IF 	eState = 0 THEN // eDisabled := 0,	
	sStateDesc := 'Wyłączona';
ELSIF 	eState = 1 THEN // eAborted := 1,
	sStateDesc := 'Bezpieczne zatrzymanie';
ELSIF 	eState = 2 THEN // eAborting := 2,  
	sStateDesc := 'Bezpieczne zatrzymywanie';
ELSIF 	eState = 3 THEN // eError := 3,	
	sStateDesc := 'Błąd';
ELSIF 	eState = 4 THEN // eResetting := 4,	
	sStateDesc := 'Resetowanie';
ELSIF 	eState = 5 THEN // eManualMovement := 5, 
	sStateDesc := 'Tryb serwisowy';
ELSIF 	eState = 6 THEN // eHoming := 6,
	sStateDesc := 'Bazowanie';
ELSIF 	eState = 7 THEN // eHomingDone := 7,
	sStateDesc := 'Koniec bazowania';	
ELSIF 	eState = 8 THEN // ePreparingToReady := 8,	
	sStateDesc := 'Przygotowanie do gotowości';
ELSIF 	eState = 9 THEN // ePreparingToDisable := 9,
	sStateDesc := 'Przygotowanie do wyłączenia';	
ELSIF 	eState = 10 THEN // eReady	:= 10,
	sStateDesc := 'Gotowa';	
ELSIF 	eState = 11 THEN // eStopping := 11,
	sStateDesc := 'Zatrzymywanie';	
ELSIF 	eState = 12 THEN // eStarting := 12,
	sStateDesc := 'Uruchamianie';  
ELSIF 	eState = 13 THEN // eRunning := 13		
	sStateDesc := 'Praca';
END_IF

IF eState = 13 OR bRun THEN
	GripperScrewer();
	BottleSorter();
	RollerScrewer();	
	EntranceGates();
	CatchStation();
	MassHeating();
	Conveyor();
	CapFeeder();
	Checker();
	Dispencer();
	DispencerLifter();
	Robot();
	Weight();
	WeightLift();
	Drag();
	DragPneum();
	LidFeeder();
	LidSealing();
	WickFeeder();
END_IF

iState := eState;

ACTION BottleSorter:

IF eBottleSorterRunningState  = 1 THEN 
	sStateDesc := 'Błąd';	
ELSIF eBottleSorterRunningState  = 2 THEN 
	sStateDesc := 'Gotowa';	
ELSIF eBottleSorterRunningState  = 3 THEN 
	sStateDesc := 'Bazowanie';	
ELSIF eBottleSorterRunningState  = 4 THEN 
	sStateDesc := 'Koniec bazowania';	
ELSIF eBottleSorterRunningState  = 5 THEN 
	sStateDesc := 'Tryb ręczny';
ELSIF eBottleSorterRunningState  = 60 THEN 
	sStateDesc := 'Przygotowanie do ruchu';	
ELSIF eBottleSorterRunningState  = 70 THEN 
	sStateDesc := 'Zamknięcie bramki lewej';	
ELSIF eBottleSorterRunningState  = 80 THEN 
	sStateDesc := 'Przejazd do pobrania';	
ELSIF eBottleSorterRunningState  = 90 THEN 
	sStateDesc := 'Zamykanie chwytaka';	
ELSIF eBottleSorterRunningState  = 100 THEN 
	sStateDesc := 'Otwarcie bramki prawej';	
ELSIF eBottleSorterRunningState  = 110 THEN 
	sStateDesc := 'Przejazd nad formatke';	
ELSIF eBottleSorterRunningState  = 120 THEN 
	sStateDesc := 'Zamknięcie bramki lewej';	
ELSIF eBottleSorterRunningState  = 130 THEN 
	sStateDesc := 'Zamknięcie docisku';	
ELSIF eBottleSorterRunningState  = 140 THEN 
	sStateDesc := 'Wkładanie opakowania';	
ELSIF eBottleSorterRunningState  = 150 THEN 
	sStateDesc := 'Otwieranie chwytaka';
ELSIF eBottleSorterRunningState  = 160 THEN 
	sStateDesc := 'Powrót do pozycji gotowości';
ELSIF eBottleSorterRunningState  = 170 THEN 
	sStateDesc := 'Wypuszczanie formatki';
		
END_IF
END_ACTION

ACTION CapFeeder:
IF eCapFeederRunningState = 1 THEN
	sStateDesc := 'Gotowy';
ELSIF eCapFeederRunningState = 2 THEN
	sStateDesc := 'Niski poziom zamknięć';
ELSIF eCapFeederRunningState = 3 THEN
	sStateDesc := 'Praca';
ELSIF eCapFeederRunningState = 4 THEN
	sStateDesc := 'Zapełniony';
END_IF
END_ACTION

ACTION CapPushing:
IF eCapPushingRunningState = 1 THEN
	sStateDesc := 'Gotowy';
ELSIF eCapPushingRunningState = 2 THEN
	sStateDesc := 'Wbijanie';
ELSIF eCapPushingRunningState = 3 THEN
	sStateDesc := 'Przyciskanie';	
ELSIF eCapPushingRunningState = 4 THEN
	sStateDesc := 'Wbito';		
ELSIF eCapPushingRunningState = 5 THEN
	sStateDesc := 'Podnoszenie';									
END_IF
END_ACTION

ACTION CatchStation:
IF eCatchRunningState = 1 THEN
	sStateDesc := 'Błąd';
ELSIF eCatchRunningState = 2 THEN
	sStateDesc := 'Tryb serwisowy';
ELSIF eCatchRunningState = 4 THEN
	sStateDesc := 'Bazowanie';	
ELSIF eCatchRunningState = 5 THEN
	sStateDesc := 'Koniec bazownia';		
ELSIF eCatchRunningState = 6 THEN
	sStateDesc := 'Gotowość';			
ELSIF eCatchRunningState = 7 THEN
	sStateDesc := 'Chwytanie';				
ELSIF eCatchRunningState = 8 THEN
	sStateDesc := 'Chwycono';					
ELSIF eCatchRunningState = 9 THEN
	sStateDesc := 'Przygotowanie do wyłączenia';	
ELSIF eCatchRunningState = 10 THEN
	sStateDesc := 'Nie chwycono';					
END_IF
END_ACTION

ACTION Checker:
IF eCheckerRunningState = 1 THEN
	sStateDesc := 'Blad';
ELSIF eCheckerRunningState = 2 THEN
	sStateDesc := 'Tryb serwisowy';	
ELSIF eCheckerRunningState = 3 THEN
	sStateDesc := 'Bazowanie';		
ELSIF eCheckerRunningState = 4 THEN
	sStateDesc := 'Koniec bazowania';			
ELSIF eCheckerRunningState = 5 THEN
	sStateDesc := 'Gotowa';				
ELSIF eCheckerRunningState = 6 THEN
	sStateDesc := 'Formatka';		
ELSIF eCheckerRunningState = 7 THEN
	sStateDesc := 'Butelka';	
ELSIF eCheckerRunningState = 8 THEN
	sStateDesc := 'Platynka OK';	
ELSIF eCheckerRunningState = 9 THEN
	sStateDesc := 'Nasadka OK';	
ELSIF eCheckerRunningState = 10 THEN
	sStateDesc := 'Nasadka NOK.';		
ELSIF eCheckerRunningState = 11 THEN
	sStateDesc := 'Przyg. do wył.';		
					
END_IF
END_ACTION

ACTION Conveyor:
(*IF eConveyorRunningState = 0 THEN //Wyłączona
	sStateDesc := 'Wyłączona';
ELSIF eConveyorRunningState = 1 THEN //Błąd
	sStateDesc := 'Bład';
ELSIF eConveyorRunningState = 2 THEN //Tryb serwisowy
	sStateDesc := 'Tryb serwisowy';	
ELSIF eConveyorRunningState = 3 THEN //Bazowanie
	sStateDesc := 'Bazowanie';		
ELSIF eConveyorRunningState = 4 THEN //Koniec bazowania
	sStateDesc := 'Koniec bazowanie';	
ELSIF eConveyorRunningState = 5 THEN //gotowość
	sStateDesc := 'Gotowa';	
ELSIF eConveyorRunningState = 6 THEN //Zatrzymywanie
	sStateDesc := 'Zatrzymywanie';	
ELSIF eConveyorRunningState = 7 THEN //Startowanie
	sStateDesc := 'Startowanie';	
ELSIF eConveyorRunningState = 8 THEN //Praca
	sStateDesc := 'Praca';				
END_IF


*)
(*
IF eConveyorRunningState = 0 THEN //Wyłączona
	sStateDesc := 'Wyłączona 123';
ELSIF eConveyorRunningState = 1 THEN //Błąd
	sStateDesc := 'Bezp. zatrzymana';
ELSIF eConveyorRunningState = 2 THEN //Tryb serwisowy
	sStateDesc := 'Bezp. zatrzymywanie';	
ELSIF eConveyorRunningState = 3 THEN //Bazowanie
	sStateDesc := 'Błąd';		
ELSIF eConveyorRunningState = 4 THEN //Koniec bazowania
	sStateDesc := 'Resetowanie błędów';	
ELSIF eConveyorRunningState = 5 THEN //gotowość
	sStateDesc := 'Tryb ręczny';	
ELSIF eConveyorRunningState = 6 THEN //Zatrzymywanie
	sStateDesc := 'Bazowanie';	
ELSIF eConveyorRunningState = 7 THEN //Startowanie
	sStateDesc := 'Koniec bazowania';	
ELSIF eConveyorRunningState = 8 THEN //Praca
	sStateDesc := 'Przyg. do wył.';	
	*)
IF eConveyorRunningState = 10 THEN //Startowanie
	sStateDesc := 'Gotowośc';	
ELSIF eConveyorRunningState = 11 THEN //Praca
	sStateDesc := 'Zatrzymywanie';	
ELSIF eConveyorRunningState = 12 THEN //Praca
	sStateDesc := 'Uruchamianie';	
ELSIF eConveyorRunningState = 13 THEN //Praca
	sStateDesc := 'Praca';

	
END_IF
END_ACTION

ACTION Dispencer:
IF eDispencerRunningState = 5 THEN
	sStateDesc := 'Gotowa';	
		ic3		:= ic3+1;		
ELSIF eDispencerRunningState = 6 THEN
	sStateDesc := 'Przyg. dozy';		
ELSIF eDispencerRunningState = 7 THEN
	sStateDesc := '1 faza';	
ELSIF eDispencerRunningState = 8 THEN
	sStateDesc := '2 faza';	
ELSIF eDispencerRunningState = 9 THEN
	sStateDesc := '3 faza';	
ELSIF eDispencerRunningState = 10 THEN
	sStateDesc := 'Koniec dozy';	
ELSIF eDispencerRunningState = 11 THEN
	sStateDesc := 'Podsys';	
ELSIF eDispencerRunningState = 12 THEN
	sStateDesc := 'Koniec pods.';	
ELSIF eDispencerRunningState = 13 THEN
	sStateDesc := 'Zasysanie';				
ELSIF eDispencerRunningState = 14 THEN
	sStateDesc := 'Podnoszenie';	
ELSIF eDispencerRunningState = 15 THEN
	sStateDesc := 'Przerywanie';			
ELSIF eDispencerRunningState = 16 THEN
	sStateDesc := 'Przyg. do wył.';	
ELSIF eDispencerRunningState = 17 THEN
	sStateDesc := 'Przeciąganie';
ELSIF eDispencerRunningState = 18 THEN
	sStateDesc := 'Przyg. do mycia';
ELSIF eDispencerRunningState = 19 THEN
	sStateDesc := 'Gotowy do mycia';
ELSIF eDispencerRunningState = 20 THEN
	sStateDesc := 'Mycie';
ELSIF eDispencerRunningState = 21 THEN
	sStateDesc := 'Koniec mycia';		
END_IF

i   := eDispencerRunningState;
END_ACTION

ACTION DispencerLifter:
IF eDispencerLifterRunningState = 1 THEN
	sStateDesc := 'Blad';
ELSIF eDispencerLifterRunningState = 2 THEN
	sStateDesc := 'Tryb serwisowy';	
ELSIF eDispencerLifterRunningState = 3 THEN
	sStateDesc := 'Bazowanie';		
ELSIF eDispencerLifterRunningState = 4 THEN
	sStateDesc := 'Koniec bazowania';			
ELSIF eDispencerLifterRunningState = 5 THEN
	sStateDesc := 'Gotowa';				
ELSIF eDispencerLifterRunningState = 6 THEN
	sStateDesc := 'Przyg. dozy';		
ELSIF eDispencerLifterRunningState = 7 THEN
	sStateDesc := '1 faza';	
ELSIF eDispencerLifterRunningState = 8 THEN
	sStateDesc := '2 faza';	
ELSIF eDispencerLifterRunningState = 9 THEN
	sStateDesc := '3 faza';	
ELSIF eDispencerLifterRunningState = 10 THEN
	sStateDesc := 'Koniec dozy';	
ELSIF eDispencerLifterRunningState = 11 THEN
	sStateDesc := 'Zasysanie';	
ELSIF eDispencerLifterRunningState = 12 THEN
	sStateDesc := 'Podnoszenie';	
ELSIF eDispencerLifterRunningState = 13 THEN
	sStateDesc := 'Wylaczanie';				
ELSIF eDispencerLifterRunningState = 14 THEN
	sStateDesc := 'Przyg. do wył.';	
ELSIF eDispencerLifterRunningState = 15 THEN
	sStateDesc := 'Przeciąganie';			
ELSIF eDispencerLifterRunningState = 16 THEN
	sStateDesc := 'Podsysanie';	
ELSIF eDispencerLifterRunningState = 17 THEN
	sStateDesc := 'Koniec podsysania';		
END_IF
END_ACTION

ACTION Drag:
IF eFormsDragingRunningState = 1 THEN 
	sStateDesc := 'Bład';
ELSIF eFormsDragingRunningState  = 2 THEN 
	sStateDesc := 'Gotowość';	
ELSIF eFormsDragingRunningState  = 3 THEN 
	sStateDesc := 'Tryb serwisowy';	
ELSIF eFormsDragingRunningState  = 4 THEN 
	sStateDesc := 'Przygotowanie do ruchu';	
ELSIF eFormsDragingRunningState  = 5 THEN 
	sStateDesc := 'Bazowanie';	
ELSIF eFormsDragingRunningState  = 6 THEN 
	sStateDesc := 'Koniec bazowania';	
ELSIF eFormsDragingRunningState  = 7 THEN 
	sStateDesc := 'Podnoszenie';	
ELSIF eFormsDragingRunningState  = 8 THEN 
	sStateDesc := 'Przyg. do przec.';	
ELSIF eFormsDragingRunningState  = 9 THEN 
	sStateDesc := 'Przeciąganie';	
ELSIF eFormsDragingRunningState  = 10 THEN 
	sStateDesc := 'Koniec Przec.';	
ELSIF eFormsDragingRunningState  = 11 THEN 
	sStateDesc := 'Zakańczanie przec.';	
ELSIF eFormsDragingRunningState  = 12 THEN 
	sStateDesc := 'Koniec zakań. przec.';	
ELSIF eFormsDragingRunningState  = 13 THEN 
	sStateDesc := 'Opuszczanie';	
ELSIF eFormsDragingRunningState  = 14 THEN 
	sStateDesc := 'Przeciągniete';	
ELSIF eFormsDragingRunningState  = 15 THEN 
	sStateDesc := 'Koniec cyklu';	
			
END_IF
END_ACTION

ACTION DragPneum:
IF eFormsDragingPneumRunningState= 1 THEN 
	sStateDesc := 'Bład';
ELSIF eFormsDragingPneumRunningState  = 2 THEN 
	sStateDesc := 'Gotowość';	
ELSIF eFormsDragingPneumRunningState  = 3 THEN 
	sStateDesc := 'Tryb serwisowy';	
ELSIF eFormsDragingPneumRunningState  = 4 THEN 
	sStateDesc := 'Przygotowanie do ruchu';	
ELSIF eFormsDragingPneumRunningState  = 5 THEN 
	sStateDesc := 'Bazowanie';	
ELSIF eFormsDragingPneumRunningState  = 6 THEN 
	sStateDesc := 'Koniec bazowania';	
ELSIF eFormsDragingPneumRunningState  = 7 THEN 
	sStateDesc := 'Podnoszenie';	
ELSIF eFormsDragingPneumRunningState  = 8 THEN 
	sStateDesc := 'Przyg. do przec.';	
ELSIF eFormsDragingPneumRunningState  = 9 THEN 
	sStateDesc := 'Przeciąganie';	
ELSIF eFormsDragingPneumRunningState  = 10 THEN 
	sStateDesc := 'Koniec Przec.';	
ELSIF eFormsDragingPneumRunningState  = 11 THEN 
	sStateDesc := 'Korekta pozycji';	
ELSIF eFormsDragingPneumRunningState  = 12 THEN 
	sStateDesc := 'Koniec korekty';	
ELSIF eFormsDragingPneumRunningState  = 13 THEN 
	sStateDesc := 'Opuszczanie';	
ELSIF eFormsDragingPneumRunningState  = 14 THEN 
	sStateDesc := 'Przeciągniete';	
ELSIF eFormsDragingPneumRunningState  = 15 THEN 
	sStateDesc := 'Koniec cyklu';					
END_IF
END_ACTION

ACTION EntranceGates:
IF eEntranceGatesRunningState = 1 THEN
	sStateDesc := 'Błąd';
ELSIF eEntranceGatesRunningState = 2 THEN
	sStateDesc := 'Tryb serwisowy';
ELSIF eEntranceGatesRunningState = 4 THEN
	sStateDesc := 'Bazowanie';	
ELSIF eEntranceGatesRunningState = 5 THEN
	sStateDesc := 'Koniec bazownia';		
ELSIF eEntranceGatesRunningState = 6 THEN
	sStateDesc := 'Gotowość';			
ELSIF eEntranceGatesRunningState = 8 THEN
	sStateDesc := 'Wjazd 2 ';				
ELSIF eEntranceGatesRunningState = 9 THEN
	sStateDesc := 'Wjazd 1';					
ELSIF eEntranceGatesRunningState = 11 THEN
	sStateDesc := 'Czekanie';						
ELSIF eEntranceGatesRunningState = 12 THEN
	sStateDesc := 'Wyjazd 2';							
ELSIF eEntranceGatesRunningState = 13 THEN
	sStateDesc := 'Wyjazd 1';	
ELSIF eEntranceGatesRunningState = 14 THEN
	sStateDesc := 'Blokowanie';	
ELSIF eEntranceGatesRunningState = 15 THEN
	sStateDesc := 'Otwieranie';	
ELSIF eEntranceGatesRunningState = 16 THEN
	sStateDesc := 'Otwarty';	
ELSIF eEntranceGatesRunningState = 17 THEN
	sStateDesc := 'Przygotowanie do gotowości';	
ELSIF eEntranceGatesRunningState = 18 THEN
	sStateDesc := 'Przygotowanie do wyłączenia';	
ELSIF eEntranceGatesRunningState = 19 THEN
	sStateDesc := 'Przeciąganie do środka';	
ELSIF eEntranceGatesRunningState = 20 THEN
	sStateDesc := 'Przeciągnięto do środka';			
END_IF
END_ACTION

ACTION GripperScrewer:
IF eGripperScrewerRunningState = 1 THEN
	sStateDesc := 'Gotowa';
ELSIF eGripperScrewerRunningState = 2 THEN
	sStateDesc := 'Przejazd do wbijania';
ELSIF eGripperScrewerRunningState = 3 THEN
	sStateDesc := 'Przejazd do zakrecania';	
ELSIF eGripperScrewerRunningState = 4 THEN
	sStateDesc := 'Wcisnieto';		
ELSIF eGripperScrewerRunningState = 5 THEN
	sStateDesc := 'Szukanie gwintu';			
ELSIF eGripperScrewerRunningState = 6 THEN
	sStateDesc := 'Zakrecanie';				
ELSIF eGripperScrewerRunningState = 7 THEN
	sStateDesc := 'Podnoszenie';					
ELSIF eGripperScrewerRunningState = 8 THEN
	sStateDesc := 'Zakrecono';						
ELSIF eGripperScrewerRunningState = 9 THEN
	sStateDesc := 'Niezakręcono';							
ELSIF eGripperScrewerRunningState = 10 THEN
	sStateDesc := 'Przytrzymywanie';			
END_IF
END_ACTION

ACTION LidFeeder:
IF eLidFeederRunningState = 1 THEN
	sStateDesc := 'Blad';
ELSIF eLidFeederRunningState = 2 THEN
	sStateDesc := 'Tryb serwisowy';	
ELSIF eLidFeederRunningState = 3 THEN
	sStateDesc := 'Bazowanie';		
ELSIF eLidFeederRunningState = 4 THEN
	sStateDesc := 'Koniec bazowania';			
ELSIF eLidFeederRunningState = 5 THEN
	sStateDesc := 'Nagrzewanie';				
ELSIF eLidFeederRunningState = 6 THEN
	sStateDesc := 'Gotowa';		
ELSIF eLidFeederRunningState = 7 THEN
	sStateDesc := 'Zasysanie';	
ELSIF eLidFeederRunningState = 8 THEN
	sStateDesc := 'Nakładanie';	
ELSIF eLidFeederRunningState = 9 THEN
	sStateDesc := 'Nakładanie 2';	
ELSIF eLidFeederRunningState = 10 THEN
	sStateDesc := 'Zgrzewanie';	
ELSIF eLidFeederRunningState = 11 THEN
	sStateDesc := 'Odlożona';	
ELSIF eLidFeederRunningState = 12 THEN
	sStateDesc := 'Podnoszenie';	
ELSIF eLidFeederRunningState = 13 THEN
	sStateDesc := 'Przyg.do wyłączenia';						
END_IF
END_ACTION

ACTION LidSealing:

IF eLidSealingRunningState = 1 THEN
	sStateDesc := 'Nagrzewanie';
ELSIF eLidSealingRunningState = 2 THEN
	sStateDesc := 'Gotowa';	
ELSIF eLidSealingRunningState = 3 THEN
	sStateDesc := 'Zgrzewanie';		
ELSIF eLidSealingRunningState = 4 THEN
	sStateDesc := 'Grzanie';			
ELSIF eLidSealingRunningState = 5 THEN
	sStateDesc := 'Zgrzano';				
ELSIF eLidSealingRunningState = 6 THEN
	sStateDesc := 'Podnoszenie';							
END_IF
END_ACTION

ACTION MassHeating:
IF eMassHeatingRunningState = 1 THEN //Grzanie
	sStateDesc := 'Grzanie';
ELSIF eMassHeatingRunningState = 2 THEN //Gotowość
	sStateDesc := 'Utrzymywanie temp.';	
ELSIF eMassHeatingRunningState = 3 THEN //Chłodzenie
	sStateDesc := 'Chłodzenie';					
END_IF
END_ACTION

ACTION Robot:
IF eCapFeederRobotRunningState = 1 THEN
	sStateDesc := 'Pobieranie';
ELSIF eCapFeederRobotRunningState = 2 THEN
	sStateDesc := 'Pobrano';
ELSIF eCapFeederRobotRunningState = 3 THEN
	sStateDesc := 'Odkładanie';	
ELSIF eCapFeederRobotRunningState = 4 THEN
	sStateDesc := 'Pobrano';		
ELSIF eCapFeederRobotRunningState = 5 THEN
	sStateDesc := 'Odrzucanie';			
ELSIF eCapFeederRobotRunningState = 6 THEN
	sStateDesc := 'Odrzucono';				
ELSIF eCapFeederRobotRunningState = 7 THEN
	sStateDesc := 'Do start Inkjet';	
ELSIF eCapFeederRobotRunningState = 8 THEN
	sStateDesc := 'Start Inkjet';		
ELSIF eCapFeederRobotRunningState = 9 THEN
	sStateDesc := 'Do stop Inkjet';		
ELSIF eCapFeederRobotRunningState = 10 THEN
	sStateDesc := 'Stop Inkjet';		
ELSIF eCapFeederRobotRunningState = 11 THEN
	sStateDesc := 'Przerywanie';		
ELSIF eCapFeederRobotRunningState = 12 THEN
	sStateDesc := 'Powrót do gotowości';		
ELSIF eCapFeederRobotRunningState = 13 THEN
	sStateDesc := 'Pobieranie po Estopie';						
END_IF
END_ACTION

ACTION RollerScrewer:
(*IF eRollerScrewerRunningState = 1 THEN
	sStateDesc := 'Gotowa';
ELSIF eRollerScrewerRunningState = 2 THEN
	sStateDesc := 'Wciskanie';
ELSIF eRollerScrewerRunningState = 3 THEN
	sStateDesc := '';	
ELSIF eRollerScrewerRunningState = 4 THEN
	sStateDesc := 'Wcisnieto';		
ELSIF eRollerScrewerRunningState = 5 THEN
	sStateDesc := 'Szukanie gwintu';			
ELSIF eRollerScrewerRunningState = 6 THEN
	sStateDesc := 'Zakrecanie';				
ELSIF eRollerScrewerRunningState = 7 THEN
	sStateDesc := 'Podnoszenie';					
ELSIF eRollerScrewerRunningState = 8 THEN
	sStateDesc := 'Zakrecono';						
ELSIF eRollerScrewerRunningState = 9 THEN
	sStateDesc := 'Niezakręcono';							
ELSIF eRollerScrewerRunningState = 10 THEN
	sStateDesc := 'Przytrzymywanie';			
END_IF

*)
END_ACTION

ACTION Weight:
IF  eWeightRunningState = 1 THEN
	sStateDesc := 'Gotowa';	
ELSIF eWeightRunningState = 2 THEN
	sStateDesc := 'Ważenie';		
ELSIF eWeightRunningState = 3 THEN
	sStateDesc := 'Koniec ważenia';					
END_IF
END_ACTION

ACTION WeightLift:
IF  eWeightLiftRunningState	 = 10 THEN
	sStateDesc := 'Gotowa';	
ELSIF eWeightLiftRunningState	= 20 THEN
	sStateDesc := 'Przyg do magazynowania formatek';		
ELSIF eWeightLiftRunningState	 = 30 THEN
	sStateDesc := 'Czekanie na formatki';		
ELSIF eWeightLiftRunningState	 = 40 THEN
	sStateDesc := 'Rozpoczęcie ważenia';		
ELSIF eWeightLiftRunningState	 = 50 THEN
	sStateDesc := 'Ważenie';		
ELSIF eWeightLiftRunningState	 = 60 THEN
	sStateDesc := 'Opuszczanie wideł';		
ELSIF eWeightLiftRunningState	 = 70 THEN
	sStateDesc := 'Wypuszczanie formatek';		
ELSIF eWeightLiftRunningState	 = 80 THEN
	sStateDesc := 'Cykl skończony';			
END_IF
END_ACTION

ACTION Wheel:
(*IF eWheelRunningState = 1 THEN
	sStateDesc := 'Blad';
ELSIF eWheelRunningState = 2 THEN
	sStateDesc := 'Tryb serwisowy';	
ELSIF eWheelRunningState = 3 THEN
	sStateDesc := 'Bazowanie';		
ELSIF eWheelRunningState = 4 THEN
	sStateDesc := 'Koniec bazowania';			
ELSIF eWheelRunningState = 5 THEN
	sStateDesc := 'Gotowa';				
ELSIF eWheelRunningState = 6 THEN
	sStateDesc := 'Obracanie';		
ELSIF eWheelRunningState = 7 THEN
	sStateDesc := 'Koniec obracania';	
ELSIF eWheelRunningState = 8 THEN
	sStateDesc := 'Przerywanie';	
ELSIF eWheelRunningState = 9 THEN
	sStateDesc := 'Obracanie 2';	
ELSIF eWheelRunningState = 10 THEN
	sStateDesc := 'Przygtowanie go obr.';						
END_IF
*)
END_ACTION

ACTION WickFeeder:
IF eWickFeederRunningState = 1 THEN
	sStateDesc := 'Blad';
ELSIF eWickFeederRunningState = 2 THEN
	sStateDesc := 'Tryb serwisowy';	
ELSIF eWickFeederRunningState = 3 THEN
	sStateDesc := 'Bazowanie';		
ELSIF eWickFeederRunningState = 4 THEN
	sStateDesc := 'Koniec bazowania';			
ELSIF eWickFeederRunningState = 5 THEN
	sStateDesc := 'Nagrzewanie';				
ELSIF eWickFeederRunningState = 6 THEN
	sStateDesc := 'Gotowa';		
ELSIF eWickFeederRunningState = 7 THEN
	sStateDesc := 'Zasysanie';	
ELSIF eWickFeederRunningState = 8 THEN
	sStateDesc := 'Nakładanie';	
ELSIF eWickFeederRunningState = 9 THEN
	sStateDesc := 'Nakładanie 2';	
ELSIF eWickFeederRunningState = 10 THEN
	sStateDesc := 'Zgrzewanie';	
ELSIF eWickFeederRunningState = 11 THEN
	sStateDesc := 'Odlożona';	
ELSIF eWickFeederRunningState = 12 THEN
	sStateDesc := 'Podnoszenie';	
ELSIF eWickFeederRunningState = 13 THEN
	sStateDesc := 'Przyg.do wyłączenia';						
END_IF
END_ACTION

END_FUNCTION_BLOCK

// ---- POUs/FB/FB_ROPPFeeder.TcPOU
(*
Nazwa:			FB_ROPPFeeder
Opis:			Sorter nasadek i podajnik nasadek z podnośnikiem JIESANG
Wersja:			v0.1
Data:			2022-07-07
Autor:			DJA
Urzadzenia:		Silnik sortera, podnośnik JIESANG, Wydmuch, czujniki zapełnienia rękawa
Konfiguracja:	
Info:
-poprawiona wersja sortera względem poprzedniej, przerobione na aktualny standard State i RunningState
*)


FUNCTION_BLOCK FB_ROPPFeeder
VAR_INPUT
	
	bEnable						: BOOL;					//Zezowlenie na pracę stacji sprawdzania
	bEStop						: BOOL;					//Stop Awaryjny nieaktywny
	bRun						: BOOL;					//
	bHoming						: BOOL;					//Zezwolenie na wykonanie bazowania i pozycjonowania stacji sprawdzania
	bHeightSet					: BOOL;					//Bit do bazowania stacji na ustaloną wysokość 
	bIgnoreError				: BOOL;					//Ignorowania błędów cyklu pracy
	bReset						: BOOL;					//Reset błędu, jeśli w stanie "eError"

	bConveyorOKSensor			: BOOL;					
	bConveyorNOKSensor			: BOOL;				
	bAirOKSensor				: BOOL;					// 
	bCapsWheelLevelSensor		: BOOL;					// Czujnik poziomu
	bCapsLevelSensor			: BOOL;					// Czujnik poziomu
	bCapsSleeveSensor			: BOOL;					// 

	iTimeDelayOn				: INT; 					//Czas na właczenie silnika sortera po zaniku sygnału przepełnienia z rękawa
	iTimeDelayOff				: INT; 					// Czas na wylączenie silnika sortera po wykryciu sygnału przepełnienia z rękawa sortera
	iTimeToEmptySleeveError		: INT;					// Czas do włączenia alrmu pustego rękawa
	InEngineVelocityCV 			: UDINT;		
	InEngineSTW 				: UINT; 				// Statusword transportera wejściowo wyjściowego
	IbEngineWcState				: BOOL; 				// Statusword transportera wejściowo wyjściowego

	_HEIGHTMOTOR_ 				: BOOL;
	lrHeightMotorSV				: LREAL;				// Zadana wysokość
	udiHeightMotorEncoderCV		: UDINT;				// Ilość impulsów z modułu enkoderowego
	bHeightEncoderSetCDone		: BOOL;					// Zerowanie enkodera wykonane
	rHeightMotorPositionOffset 	: REAL;					// Wysokość bazowani podnośnika
	lrMaxHeight					: LREAL;				// Maksymalna wysokość podnośnika chwytaka
	lrMinHeight					: LREAL;				// Minimalna wysokość podnośnika chwytaka

	bManualMovement				: BOOL; 				//Uruchomienie trybu ruchów ręcznych
	udiStationIndex				: UDINT;				// Indywidualny numer stacji
	sStationName				: STRING;				// Nazwa stacji	
END_VAR

VAR_OUTPUT
	eState						: E_Station;			// Aktualny stan stacju
	eRunningState				: E_CapFeederState;		// Stan pracy stacji
	eRunningStateBeforeEstop	: E_CapFeederState;  	// Stan przed Estope
	bError						: BOOL;					// Błąd stacji
	udiErrorID					: UDINT;				// Nr blędu przeciągania formatek
	sErrorDescription			: STRING(200);			// Opis błędu
	sErrorDescription2			: STRING(200);			// Opis błędu
	sErrorStationName			: STRING;				// Nazwa stacj
	udiStationID				: UDINT;				// Nr stacji

	bHeightMotorUp				: BOOL;					//Sterowanie silnikiem podnośnika  - RUCH W GÓRĘ
	bHeightMotorDown			: BOOL;					//Sterowanie silnikiem podnośnika  - RUCH W DÓŁ
	udiHeightMotorEncoderSetCV	: UDINT;		
	bHeightEncoderSetC			: BOOL;					// Zerowanie enkodera
	lrHeightMotorCV				: LREAL;				// Aktualna pozycja podnośnika

	QnEngineVelocitySV 			: UDINT; 				// Nastawa prędkości
	QnEngineCTW 				: UINT;  				// Controlword transportera we/wy	
	bSorterVibrator				: BOOL; 	
	bSorterAir 					: BOOL; 				
	bSorterAir2					: BOOL; 				
	bConveyorStart				: BOOL; 				
	bConveyorStop				: BOOL; 	
	
	bHomingNeeded				: BOOL;					// Wymagane ponowne bazowanie (blad podczas bazowania lub stop awaryjny)
	bHomingDone					: BOOL;					// Stacja zbazowana 
	bCycleDone					: BOOL;					// Sygnał o zakończeniu cyklu
	bCycleNotDone				: BOOL;					// Sygnał o niezakończonym cyklu
	tCycleTime					: TIME;	 				// Czas cyklu 
	sWarningDescription			: STRING;
	bWarning1					: BOOL;
	udiWarningID				: UDINT;
	
END_VAR

VAR_IN_OUT
	bManualHeightMotorUp		: BOOL;					//Ruch ręczny podnośnika stacji w górę
	bManualHeightMotorDown		: BOOL;					//Ruch ręczny podnośnika stacji w dół
	bManualSorterEngine			: BOOL;					//
	bManualSorterVibrator		: BOOL;					//
	bManualSorterAir 			: BOOL;					//
	bManualSorterAir2			: BOOL;					//
	bManualConveyorStart		: BOOL;					//
	bManualConveyorStop			: BOOL;					//
END_VAR

VAR
	i							:	INT;
	aBufferedSensorValue		:	ARRAY[0..50] OF BOOL;	
	rtOutSensor					:	R_TRIG;

	// State
	eLastState					: E_Station;			//Stan ogólny bloku
	eLastStateTemp				: E_Station;			//Stan ogólny bloku
	eLastRunningState			: E_CapFeederState;		//Stan podbloku
	eLastRunningStateTemp		: E_CapFeederState;		//Stan podbloku

	fbHeightMotorEncoder		: FB_JiesangActuatorEncoderModul;				// Blok enkodera podnośnika chwytaka stabilizującego pod zakręcarką	
	bHeightMotorEncoderCounterReset						:BOOL; 				// Sygnał resetu enkodera
	lrLastHeightMotorPositionCV		: LREAL;				// Pozycja podnośnika w poprzednim cyklu programu
	bHeightMotorEncoderHomed	: BOOL;					// Informacja od enkodera że jest zbazowany		
	bStateError					: BOOL;
	
	tofHeightMotorDown			: TOF;					// Opóźnienie ruchu w dół, żeby nie przeciązać rozruchem układu
	rtEncoderHomed				: R_TRIG;				// Bit zakończenia enkodera
		
	tonHeightNoChange			: TON; 					// Timer wykrycia braku ruchu siłownika zmiany wysokości stacji
	tonHeightNoChangeTime		: TON; 					// Timer wykrycia braku ruchu siłownika zmiany wysokości stacji
	
	tonLimitPosMinReachedDelay	: TON;					// Timer osoiągniecia minimalnej wyskości 
	tonLimitPosMaxReachedDelay	: TON;					// Timer osiągnięcia maksymalnej wyskości
	tonSortingEngineOn			: TON;					// Opóźnienie po załączeniu napędu
	tonSortingEngineOff			: TON;					// Opóźnienie wyłączenia napędu
	tonSleeveFullEngineOn		: TON;					// Czas załączenia napędu po wykrciu braku nasadek
	tonEngineBlocked			: TON;					// Zablokowany silnik	
	rtCapSorterSensor			: R_TRIG;				// Triger
	tonTryUnblockWheel			: TON;					// Czas ruchu falownika w drugą stronę
	tofCapFeederSorterCapSensor	: TOF;					// Opóźnienie sygnału z czujnika obecności nasadki ultradzwiek
	tonCapFeederSorterCapSensor	: TON;					// Opóźnienie sygnału z czujnika obecności nasadki ultradźwięk
	tonAirBeforeStart			: TON;					// Czasówka opóźeniani przedmuchu
	tonAirBeforeStart2			: TON;					// Czasówka opóźeniani przedmuchu
	tonAirAfterStop				: TON;					// Czasówka przedmuchu po zatrzymaniu
	tonStoppingTime				: TON;					// Czasówka zbyt długiego zatrzymawania

	
	tonErrorHeightChange		: TON; 					// Timer błędu zacięcia się podnośnika
	tonEmptySleeveError			: TON;					// Timer pustego rękawa
	tonMaxHeightError			: TON;					// Timer ustawienia zbyt dużej wysokości stacji
	tonMinHeightError			: TON;					// Timer ustawienia zbyt małej wysokości stacji
	tonCycleTimer				: TON;					// Czasówka cyklu
	rtrigCycleTimerRead			: R_TRIG;				// Trigger do statystyk cyklu 
	
	tonSorterEngineError: TON;

	TimerOn: TON;
	TimerOff: TON;
	bImpOn: BOOL;
	rtCapFeederSorterCapSensor: R_TRIG;
	bBlowDelay: BOOL;
	tonbBlowDelay: TON;
	
	fbInverter: FB_MitsubishiInverter;
	
	tonInverterError: TON;
	(*Ostrzeżenia*)
	fbbLevelSensor:	FB_InputFilter;
	(*Inne*)	
	fbbCapsWheelLevelSensor 		:	FB_InputFilter_v2;
	fbbCapsLevelSensor				:	FB_InputFilter_v2;


	tonGates1	:	TON;	//Czasówka dla szlabanów w rękawe
	tonGates2	:	TON;	//Czasówka dla szlabanów w rękawe
	tonGates3	:	TON;	//Czasówka dla szlabanów w rękawe
	tonGates4	:	TON;	//Czasówka dla szlabanów w rękawe

		
	bGates	    :	BOOL;	//Controla szłabanow w rękawe  
	bTryUnblockWheel : BOOL;
	iTryUnblockWheel : INT;
END_VAR

//Wywołanie bloczków od stacji. Ważna jest ich kolejność!!!
ACT_Limits();
ACT_HeightMotor();
ACT_ErrorHandling();

ACT_Signals();
ACT_Control();
ACT_Inverter();
ACT_Statistic();
ACT_Status();
ACT_Warnings();
aStationID();	

lrLastHeightMotorPositionCV:=lrHeightMotorCV;

ACTION ACT_Control:
	(*****Wyłączenie enable*****)
	IF NOT bEnable THEN
		IF eState <> E_Station.eDisabled AND eState <> E_Station.ePreparingToDisable THEN
				eState 				:= E_Station.ePreparingToDisable; 
		END_IF	
	END_IF

	(*****Estop*****)
	IF NOT bEstop  THEN	
		IF eState <> E_Station.eAborted AND eState <> E_Station.eAborting AND eState <> E_Station.eDisabled THEN
				eState 				:= E_Station.eAborting; 
		END_IF
	END_IF


	CASE eState OF
//--------------------------------------------------------------------------------
// Stan maszyny po wyłączeniu i przygotowanie do uruchomienia
	E_Station.eDisabled: 					// Stan nieaktywnosci (Stacja wyłączona) 
	
		IF bEnable THEN
			eState 				:= E_Station.ePreparingToReady; 
		END_IF 
		
//--------------------------------------------------------------------------------
// Stan maszyny po zatrzymaniu awaryjnym   
	E_Station.eAborted: 					// Stan bezpiecznego zatrzymania (po Abortingu) 

		IF bEStop THEN
			eState 				:= E_Station.ePreparingToReady;
		END_IF
		
//--------------------------------------------------------------------------------
// Stan maszyny naciśnieciu estopa 	
	E_Station.eAborting:                 	// Stan bezpiecznego zatrzymywania (po EStopie)

		ACT_ResetCommands();

		eState 						:=  E_Station.eAborted;  
		eRunningState				:=	E_CapFeederState.eReady;
		
//--------------------------------------------------------------------------------
// Stan masyzny po wykryciu błędu			
	E_Station.eError:                 	 	// Stan błędu 	
		
		ACT_ResetCommands();
		
		IF bReset THEN
			eState 				:= E_Station.eResetting;
			bError				:= FALSE;
		END_IF
		
//--------------------------------------------------------------------------------
// Stan masyzny po wykryciu błędu
	E_Station.eResetting:					// Stan resetowania bledu (po Errorze)
			CASE udiErrorID(*-udiStationIndex*) OF
		
				//Error 8 - Błąd falownika
				344:
					fbInverter.bReset	:= TRUE;
					bError 				:= FALSE;
				ELSE
					bError := FALSE;	
			END_CASE		
		
		IF NOT bError AND fbInverter.eState = E_Station.eReady THEN
			fbInverter.bReset	:= FALSE;	
			//{warning 'Sprawdzić błąd falownika CapFeeder'}
			udiErrorID 			:=	0;
			sErrorDescription 	:=	'';
			eState 				:=	E_Station.ePreparingToReady;
			eRunningState		:=	E_CapFeederState.eReady;
		ELSE
			eState 				:=	E_Station.eError;
		END_IF
    
//--------------------------------------------------------------------------------
// Stan ruchoow manualnych
	E_Station.eManualMovement:     			// Stan ruchów manualnych  
   
		ACT_ManualMovements();
		//Wyjście z trybu serwisowego
		IF NOT bManualMovement THEN
			
			bHeightMotorUp				:=	FALSE;
			bHeightMotorDown			:=	FALSE;
			
			eState:=E_Station.eReady;
		END_IF
		

//--------------------------------------------------------------------------------
// Stan rozpoczecia bazowania
	E_Station.eHoming:						// Stan bazowania 
		
		ACT_Homing();
		IF NOT bHoming AND NOT bHeightSet THEN
			bHeightMotorDown					:=	FALSE;
			bHeightMotorUp						:=	FALSE;
		   eState								:=	E_Station.ePreparingToReady;
		END_IF		
		
//--------------------------------------------------------------------------------
// Stan zakończenia bazowania
	E_Station.eHomingDone:                  // Stan wykonania bazowania 
	
		bHeightMotorDown					:=	FALSE;
		bHeightMotorUp						:=	FALSE;
		bHeightMotorEncoderCounterReset		:=	FALSE;
		bHomingDone							:=	TRUE;
		IF NOT bHoming AND NOT bHeightSet THEN
		   eState:=E_Station.eReady;
		END_IF
		
//--------------------------------------------------------------------------------
// Stan przygotowania do gotowości
	E_Station.ePreparingToReady:            // Stan przygotowywania do gotowosci (zawsze przed Ready)  
		
		fbInverter.bRun	:=	FALSE;
		bSorterVibrator	:=	FALSE;
		bSorterAir		:=	FALSE;
		bSorterAir2		:=	FALSE;
		bConveyorStart	:=	FALSE;
		bConveyorStop	:=	FALSE;	
		bHeightMotorUp	:=	FALSE;
		bHeightMotorDown:=	FALSE;

		eRunningState	:=	E_CapFeederState.eReady;
		eState			:=	E_Station.eReady;	
		
//-------------------------------------------------------------------------------
// Stan przygotowania do wyłączenia maszyny
	E_Station.ePreparingToDisable:          // Stan przygotowywania do nieaktywnosci (po wyłączeniu Enable) 
		
		bSorterAir			:=	FALSE;
		bHeightMotorUp		:=	TRUE;
		bHeightMotorDown	:=	FALSE;	
		IF tonHeightNoChange.Q THEN
			bHeightMotorUp			:=	FALSE;
			bHeightMotorDown		:=	FALSE;	
			eRunningState			:=	E_CapFeederState.eReady;		
			eState					:=	E_Station.eDisabled;
		END_IF	
			
//--------------------------------------------------------------------------------
// Stan gotowości
	E_Station.eReady:						// Stan gotowosci 
	
		IF bRun AND NOT bCycleDone AND NOT bCycleNotDone THEN
			eState 				:= E_Station.eStarting; 
		END_IF
		IF bHoming OR bHeightSet THEN
			bHomingDone							:=	FALSE;
			eState 								:=	E_Station.eHoming; 
		END_IF
		IF bManualMovement THEN
			//Jeśli przejście w tryb ruchów manualnych przepisz wszystkie stany siłowników sterowanych przez moduł
			//aby zapobiec ewentualnym kolizjom po wejściu w tryb serwisowy
			bManualHeightMotorUp		:= bHeightMotorUp;
			bManualHeightMotorDown		:= bHeightMotorDown;
			eState 						:= E_Station.eManualMovement; 
		END_IF
		IF NOT bRun THEN
			bCycleDone 			:= FALSE;
			bCycleNotDone 		:= FALSE;			
		END_IF
		
//--------------------------------------------------------------------------------
// Stan zatrzymywania
	E_Station.eStopping:					// Stan zatrzymywania 
		
	fbInverter.bRun	:=	FALSE;
	bSorterVibrator	:=	FALSE;
	bSorterAir		:=	TRUE;
	bSorterAir2		:=	TRUE;
	bConveyorStart	:=	FALSE;
	bConveyorStop	:=	FALSE;	
	bHeightMotorUp	:=	FALSE;
	bHeightMotorDown:=	FALSE;	
	
	IF tonStoppingTime.Q THEN
		ACT_ResetCommands();
		eRunningState							:= E_CapFeederState.eReady;
		eState									:= E_Station.eReady;
	END_IF
		
//--------------------------------------------------------------------------------
// Stan uruchomienia lini ( po eReady)
	E_Station.eStarting:                  	// Stan uruchamiania (po Ready)

		eState					 := E_Station.eRunning; 
		
//--------------------------------------------------------------------------------
// Stan wykonywania pracy
	E_Station.eRunning:               		// Stan wykonywania cyklu (po Startingu), w tym stanie osobny

		ACT_Running();
		IF NOT bRun THEN 					(*Przerywanie cyklu*)
			eState				:= E_Station.eStopping;
			//bCycleNotDone		:= TRUE;
		END_IF
		(*IF bCycleDone OR bCycleNotDone THEN (*Cykl zakończony*)
			eState 				 := E_Station.eReady;
		END_IF*)							
		
END_CASE
END_ACTION

ACTION ACT_ErrorHandling:
//OBSŁUGA BŁĘDÓW STACJI SPRAWDZANIA
//************LISTA BŁĘDÓW***************
bStateError:= (eState=E_Station.eError) OR (eState=E_Station.eResetting) OR bIgnoreError;

//************LISTA BŁĘDÓW***************

//Error 1 - podnośnik nie porusza się pomimo wysterowania 
tonErrorHeightChange(IN:=(bHeightMotorUp OR bHeightMotorDown) AND lrLastHeightMotorPositionCV=lrHeightMotorCV, PT:=T#3S);
tonEmptySleeveError(IN:=NOT bCapsSleeveSensor AND bRun, PT:=INT_TO_TIME(iTimeToEmptySleeveError)*1000); //Było 30, teraz jest z receptur
tonMaxHeightError(IN:=lrHeightMotorSV>lrMaxHeight AND NOT bHomingNeeded AND eState=E_Station.eReady,PT:=T#30S);
tonMinHeightError(IN:=lrHeightMotorSV<lrMinHeight AND NOT bHomingNeeded AND eState=E_Station.eReady,PT:=T#30S);
tonInverterError(IN:=fbInverter.bError AND NOT bStateError, PT:=T#3S);

IF (bEnable OR (eState = E_Station.ePreparingToDisable)) AND NOT bIgnoreError THEN
	
	IF tonErrorHeightChange.Q THEN
		bError:=TRUE;
		udiErrorID:=340;
		sErrorDescription:='Blokada podnośnika lub brak zasilania - sprawdź czujnik lub odblokuj mechanicznie';	
		sErrorDescription2:='';
	END_IF	
		
	//Error - Pusty rekaw sortera nasadek
	IF tonEmptySleeveError.Q THEN
		bError:=TRUE;
		udiErrorID:=341;
		sErrorDescription:='Pusty rękaw sortera - uzupełnij nasadki';
		sErrorDescription2:='';
	END_IF
	
	//Error - Bład nastaw max
	IF tonMaxHeightError.Q  THEN
		bError:=TRUE;
		udiErrorID:=342;
		sErrorDescription:='Wartość zadana wysokości jest większa od maksymalnej - zmień ustawienia w recepturze';
		sErrorDescription2:=REAL_TO_STRING(LREAL_TO_INT(lrMaxHeight));
	END_IF
	
	//Error - Bład nastaw min
	IF tonMinHeightError.Q THEN
		bError:=TRUE;
		udiErrorID:=343;
		sErrorDescription:='Wartość zadana wysokości jest mniejsza od minimalnej - zmień ustawienia w recepturze';
		sErrorDescription2:=REAL_TO_STRING(LREAL_TO_INT(lrMinHeight));
	END_IF	
	
	//Error - Bład falownika
	IF tonInverterError.Q THEN
		bError:=TRUE;
		udiErrorID:=344;
		sErrorDescription:='Błąd falownika';
		sErrorDescription2:='';
	END_IF		
	
ELSE
	bError	:=FALSE;
END_IF


//-----------------------------------------------------------------------
IF bError AND NOT bStateError THEN

	IF eLastState = eRunning THEN
		bCycleNotDone						:= TRUE;
	END_IF

	eState 									:= E_Station.eError;
END_IF


//------------------------------------------------------------------------

(*Wyświetlanie błedu na wyjściu*)
bError;

(*Przepisywanie nazwy stacji*)
sErrorStationName 							:= sStationName;

//Jezeli nie zbazowane to potrzebne bazowanie
IF NOT bHeightMotorEncoderHomed  THEN
	bHomingDone								:=	FALSE;
END_IF
END_ACTION

ACTION ACT_HeightMotor:
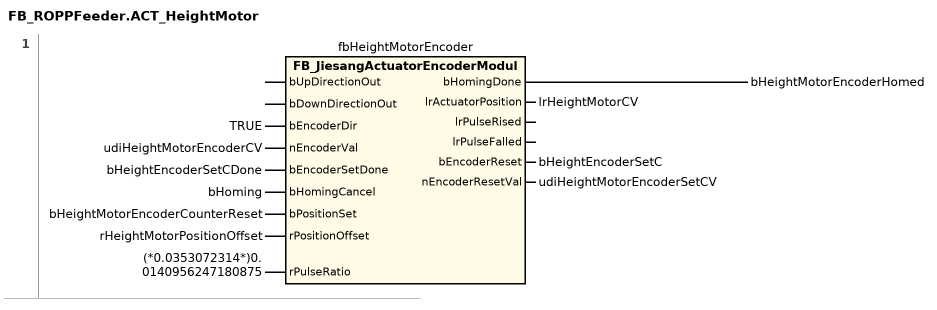
// NETWORK 1
fbHeightMotorEncoder(
    bEncoderDir := TRUE,
    nEncoderVal := udiHeightMotorEncoderCV,
    bEncoderSetDone := bHeightEncoderSetCDone,
    bHomingCancel := bHoming,
    bPositionSet := bHeightMotorEncoderCounterReset,
    rPositionOffset := rHeightMotorPositionOffset,
    rPulseRatio := (*0.0353072314*)0.0140956247180875,
    lrActuatorPosition => lrHeightMotorCV,
    bEncoderReset => bHeightEncoderSetC,
    nEncoderResetVal => udiHeightMotorEncoderSetCV); // FB_JiesangActuatorEncoderModul
bHeightMotorEncoderHomed := fbHeightMotorEncoder.bHomingDone;
END_ACTION

ACTION ACT_Homing:
//BAZOWANIE

tofHeightMotorDown(IN:=bHeightMotorDown, PT:=T#1S); //Zabezpieczenie przed zbyt szybkim przełączeniem pomiędzy Down a Up, bezpiecznieki sie palą
	
//Podnoszenie stacji do maksymalnej pozycji
IF NOT bHeightMotorEncoderHomed OR rtEncoderHomed.Q THEN
	bHeightMotorUp:=(*TRUE*) NOT tofHeightMotorDown.Q ;
	bHeightMotorDown:=FALSE;
	IF tonHeightNoChange.Q OR tonHeightNoChangeTime.Q THEN
		bHeightMotorEncoderCounterReset:=TRUE;
		bHeightMotorUp:=FALSE;
    END_IF
	//Jesli enkoder zbazowany zakończ bazowanie	
	IF rtEncoderHomed.Q  THEN
		bHeightMotorUp:=FALSE;
		bHeightMotorDown:=FALSE;
		eState:=E_Station.eHomingDone;
	END_IF		
		
//Po podniesieniu stacji opuszczanie do ustalonej wysokości
ELSIF bHeightMotorEncoderHomed THEN
	bHeightMotorEncoderCounterReset:=FALSE;
	bHeightMotorUp:=lrHeightMotorCV<=lrHeightMotorSV;
	bHeightMotorDown:=lrHeightMotorCV>=lrHeightMotorSV;
	//Kiedy stacja osiągnie wysokość zadaną
	IF ABS(lrHeightMotorCV-lrHeightMotorSV)<0.5 OR tonLimitPosMaxReachedDelay.Q OR tonLimitPosMinReachedDelay.Q THEN
		bHeightMotorDown:=FALSE;
		bHeightMotorUp:=FALSE;
		eState:=E_Station.eHomingDone;
	END_IF			
END_IF
END_ACTION

ACTION ACT_Inverter:
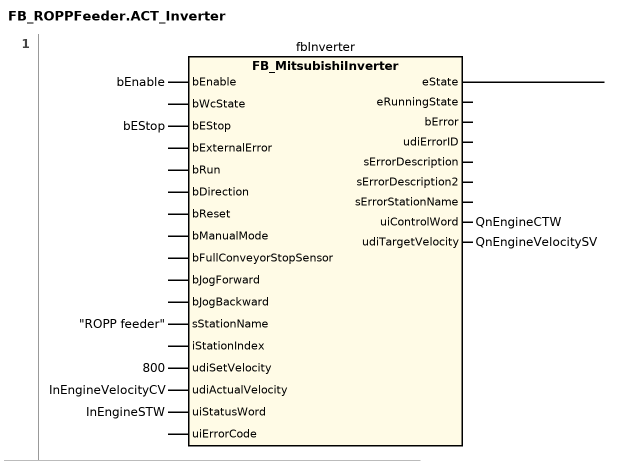
// NETWORK 1
fbInverter(
    bEnable := bEnable,
    bEStop := bEStop,
    sStationName := "ROPP feeder",
    udiSetVelocity := 800,
    udiActualVelocity := InEngineVelocityCV,
    uiStatusWord := InEngineSTW,
    uiControlWord => QnEngineCTW,
    udiTargetVelocity => QnEngineVelocitySV); // FB_MitsubishiInverter
END_ACTION

ACTION ACT_Limits:
IF iTimeToEmptySleeveError < 5 THEN
	iTimeToEmptySleeveError := 5;
END_IF
END_ACTION

ACTION ACT_ManualMovements:
//W trybie ruchów manualnych wykonuj ruchy za pomocą rozkazów manualnych
IF NOT bRun THEN
	
	fbInverter.bRun		:= bManualSorterEngine;
	bSorterVibrator		:= bManualSorterVibrator;
	bSorterAir			:= bManualSorterAir;
	bSorterAir2			:= bManualSorterAir2;
	bConveyorStart		:= bManualConveyorStart;
	bConveyorStop		:= bManualConveyorStop;
	bHeightMotorUp		:= bManualHeightMotorUp;
	bHeightMotorDown	:= bManualHeightMotorDown;

(*
*)	

END_IF


IF bHoming OR bHeightSet THEN
	eState:=E_Station.eHoming;
END_IF

IF bRun THEN	
	ACT_Running();
END_IF
//Zabezpieczenie przed kolizją stacji poprzez ruch podnośnika	
IF bHeightMotorDown AND lrHeightMotorCV<=lrMinHeight AND NOT bHoming AND NOT bHeightSet THEN
	bHeightMotorDown:=FALSE;
END_IF	

IF bHeightMotorUp AND lrHeightMotorCV>=lrMaxHeight AND NOT bHoming AND NOT bHeightSet THEN
	bHeightMotorUp:=FALSE;
END_IF
END_ACTION

ACTION ACT_ResetCommands:
//Reset komend ruchu 	


fbInverter.bRun	:=	FALSE;
bSorterVibrator	:=	FALSE;
bSorterAir		:=	FALSE;
bSorterAir2		:=	FALSE;
bConveyorStart	:=	FALSE;
bConveyorStop	:=	FALSE;	
bHeightMotorUp	:=	FALSE;
bHeightMotorDown:=	FALSE;
END_ACTION

ACTION ACT_Running:
//----------------------------------------------------------------------------------
// Obsługa podajnik zamknięc

CASE eRunningState OF
	
	//NIEGOTOWY
	E_CapFeederState.eDisabled:
		eRunningState			:=	E_CapFeederState.eReady;

	E_CapFeederState.eReady:
		iTryUnblockWheel		:=	0;
		bTryUnblockWheel		:=	FALSE;	
		fbInverter.bDirection 	:=	FALSE;
		IF bRun THEN
			eRunningState			:=E_CapFeederState.eSorting;
		END_IF
	
	E_CapFeederState.eSorting:
	

		bSorterVibrator 	:= fbbCapsWheelLevelSensor.bOUT;
		fbInverter.bRun 	:= tonAirBeforeStart.Q;
		bSorterAir 			:= TRUE;
		
		(*Zasyp*)
		bConveyorStart	:=   fbbCapsLevelSensor.bOUT;
		
		
		IF tonSortingEngineOff.Q THEN 
			eRunningState 			:=E_CapFeederState.eSleeveFull;
		END_IF
	
	E_CapFeederState.eSleeveFull:
		bSorterVibrator 	:=	FALSE;
		fbInverter.bRun		:=	FALSE;
		bConveyorStart		:=	FALSE;
		bSorterAir			:=	NOT tonAirAfterStop.Q;
		IF tonAirAfterStop.Q THEN
			IF tonSortingEngineOn.Q THEN
				eRunningState		:=E_CapFeederState.eSorting; 
			END_IF
		END_IF
	
	E_CapFeederState.eSleeveLowLevel:
	
		;
	
END_CASE
END_ACTION

ACTION ACT_Signals:
(** Timery na potrzeby bazowania**)
//Czujnik poziomu na kole
fbbCapsWheelLevelSensor	(bIN:=bCapsWheelLevelSensor , tFilterTimeOn:= T#2S, tFilterTimeOff:= T#2S, bOUT=> );
fbbCapsLevelSensor		(bIN:=NOT bCapsLevelSensor , tFilterTimeOn:= T#2S, tFilterTimeOff:= T#2S, bOUT=> );


tonAirBeforeStart		(IN:=eRunningState=E_CapFeederState.eSorting, PT:=T#1S);
tonSortingEngineOff		(IN:=((eRunningState=E_CapFeederState.eSorting OR eRunningState=E_CapFeederState.eSleeveLowLevel) AND bRun AND bCapsSleeveSensor),PT:=INT_TO_TIME(iTimeDelayOff));
tonAirAfterStop			(IN:=eRunningState=E_CapFeederState.eSleeveFull, PT:=T#2S);
tonSortingEngineOn		(IN:=((eRunningState=E_CapFeederState.eSorting OR eRunningState=E_CapFeederState.eSleeveFull) AND bRun AND NOT bCapsSleeveSensor),PT:=INT_TO_TIME(iTimeDelayOn));

rtEncoderHomed(CLK:=bHeightMotorEncoderHomed,Q=>);
tonHeightNoChange(IN:=((bHeightMotorUp OR bHeightMotorDown) AND (lrLastHeightMotorPositionCV=lrHeightMotorCV)), PT:=T#500MS); 
//tonHomingSensor(IN:=(bHomingSensor), PT:=T#100MS);
//tonHeightNoChangeTime(IN:=(eState = E_Station.eHoming OR eState = E_Station.ePreparingToDisable) AND bHeightMotorUp, PT:=T#8S); 

tonLimitPosMinReachedDelay(IN:=(lrHeightMotorCV<=lrMinHeight) AND eState=E_Station.eHoming,PT:=T#2S);
tonLimitPosMaxReachedDelay(IN:=(lrHeightMotorCV>=lrMaxHeight) AND eState=E_Station.eHoming,PT:=T#2S);
	
(** Timery używane podczas pracy stacji**)

rtCapSorterSensor(CLK:=bCapsSleeveSensor, Q=>);
//tonEngineBlocked(IN:=iTryUnblockWheel > 1500 AND bSorterEngine AND NOT bTryUnblockWheel,PT:=T#1MS); //Zablokowany silnik
tonTryUnblockWheel(IN:=bTryUnblockWheel, PT:=T#1S900MS);
tofCapFeederSorterCapSensor(IN:=tonCapFeederSorterCapSensor.Q,PT:=T#10MS); //bylo 200
tonCapFeederSorterCapSensor(IN:=bCapsSleeveSensor,PT:=T#3MS);//było 3ms

rtCapFeederSorterCapSensor(CLK:=tofCapFeederSorterCapSensor.Q,Q=>);

tonAirBeforeStart2(IN:=eRunningState=E_CapFeederState.eSorting, PT:=T#2S);


//prszesunęcie wartosci czujnika po buforu opoznenia 

FOR i:=40 TO 1 BY -1 DO
	aBufferedSensorValue[i] := aBufferedSensorValue[i-1];
END_FOR
aBufferedSensorValue[0] := bCapsSleeveSensor;

IF rtCapFeederSorterCapSensor.Q THEN
	bBlowDelay := TRUE;
	
END_IF
tonbBlowDelay(IN:=bBlowDelay,PT:=T#35MS);
IF tonbBlowDelay.Q THEN
	bBlowDelay:= FALSE;
END_IF
TimerOn (IN := NOT bImpOn, PT := T#10MS);
IF TimerOn.Q THEN
	bImpOn := TRUE;
END_IF
TimerOff (IN := bImpOn, PT := T#10MS);
IF TimerOff.Q THEN
	bImpON := FALSE;
END_IF

(** Dodatkowy timer przy zatrzymywaniu**)
tonStoppingTime( IN:= eState= E_Station.eStopping, PT:=T#2S);
END_ACTION

ACTION ACT_Statistic:
//Statystyka do zliczania czasu cyklu 
rtrigCycleTimerRead(CLK:=eRunningState=E_CapFeederState.eSleeveFull OR eRunningState=E_CapFeederState.eSleeveLowLevel);

	IF rtrigCycleTimerRead.Q THEN
		tCycleTime:=tonCycleTimer.ET;
		
	END_IF
	
tonCycleTimer(IN:=eRunningState= E_CapFeederState.eSorting , PT:=T#1D);
END_ACTION

ACTION ACT_Status:

(*Zapisywanie ostatniego stanu*)
	IF eLastStateTemp<>eState THEN
		eLastState := eLastStateTemp;
	END_IF
	eLastStateTemp := eState;
	
	IF eLastRunningStateTemp<>eRunningState THEN
		eLastRunningState := eLastRunningStateTemp;
	END_IF
	eLastRunningStateTemp := eRunningState;
(*Koniec Zapisywanie ostatniego stanu*)
END_ACTION

ACTION ACT_Warnings:
//Usrawianie warningów

//Filtrowanie czujnika ultradźwiękowego
fbbLevelSensor	(bIN:=NOT bCapsLevelSensor AND (eRunningState=E_CapFeederState.eSorting OR eRunningState=E_CapFeederState.eSleeveLowLevel OR eRunningState=E_CapFeederState.eSleeveFull) , tFilterTimeOn:= T#5S, tFilterTimeOff:=T#5S , bOUT=> );

IF fbbLevelSensor.bOUT THEN
		bWarning1						:=	TRUE;			
		udiWarningID					:=	1;
		sWarningDescription				:=	'Nieski poziom w sorterze nasadek';
ELSE
		bWarning1						:=	FALSE;			
		udiWarningID					:=	0;
		sWarningDescription				:=	'';
END_IF
END_ACTION

ACTION aStationID:
udiStationID	:=	udiStationIndex;
END_ACTION

END_FUNCTION_BLOCK

// ---- POUs/FB/FB_JiesangActuatorEncoderModul.TcPOU
(*
Nazwa:			FB_JiesangActuatorEncoder
Opis:			Obsługa podnosnika Jiesang
Wersja:			v0.1
Data:			2018-10-10
Autor:			TW
Urzadzenia:		waga HBM
Konfiguracja:	
Info: 
- podlaczenie po RS485
*)

///!!!!!WAŻNE!!!!!!!!!!
///ABY ENKODER PRACOWAŁ POPRAWNIE TASK PLC MUSI BYĆ USTAWIONY NA 3ms!!!!!!!!!
///Wynika to z faktu że korzystamy ze zwykłych wejść cyfrowych a nie szybkich liczników!!!


FUNCTION_BLOCK FB_JiesangActuatorEncoderModul
VAR_INPUT
	bUpDirectionOut:BOOL;  	//Zmienna sterownika bezpośrednio sterująca siłownikiem w górę (zlinkowana z wyjściem sterownika)
	bDownDirectionOut:BOOL;	//Zmienna sterownika bezpośrednio sterująca siłownikiem w dół (zlinkowana z wyjsciem sterownika)
	bEncoderDir	: BOOL;//Kierunek zliczania impulsów TRUE => NEGATIVE
//	bEncoderPulse:BOOL;		//Sygnał impulsów enkodera siłownika
	nEncoderVal :UDINT;		//Wartość odczytana z enkodera
	
	bEncoderSetDone:BOOL;
	bHomingCancel:BOOL;		//Anulowanie bazowania enkodera
	bPositionSet:BOOL;		//Zmienna ustawia aktualną wartości pozycji zawartą w zmiennej 'nPositionOffset'
	rPositionOffset:REAL;		//Wartość do nadpisania aktualnej pozycji po ustawieniu wejścia 'AcbtorPositionSet'
	rPulseRatio:REAL;			//Przelicznik impulsów na mm  (pokonana_odleglosc_w_mm/ilość_impulsów)
	
//	bOptionCoutingFalling : BOOL;  //Obliczenie spadania silnika
 END_VAR
VAR_OUTPUT
	bHomingDone:BOOL;
	lrActuatorPosition:LREAL:=-200;
	lrPulseRised:LREAL;
	lrPulseFalled:LREAL;
	bEncoderReset:BOOL;
	nEncoderResetVal	:UDINT;
END_VAR
VAR
	tonOffDelay	:	TON;
	rtEncoderPulse:R_TRIG;  //wykrywanie zbocza narastającego impulsu encodera
	ftEncoderPulse:F_TRIG;  //wykrywanie zbocza opadającego impulsu encodera
	rtActuatorPositionSet:R_TRIG;
	bLastDirectionUp:BOOL;
	rtHomingCancel: R_TRIG;
	nEncoderValSigned	:DINT;
	cnt : INT;
END_VAR

IF nEncoderVal.31 THEN
	nEncoderValSigned					:=  nEncoderVal - 4294967295;
ELSE
	nEncoderValSigned					:= nEncoderVal;
END_IF

IF NOT bEncoderDir THEN
	lrActuatorPosition:= rPositionOffset + TO_REAL(nEncoderValSigned) * rPulseRatio;
ELSE
	lrActuatorPosition:= rPositionOffset - TO_REAL(nEncoderValSigned) * rPulseRatio;
END_IF

//Kasowanie pozycjonowania enkodera
rtHomingCancel(CLK:=bHomingCancel,Q=>);
IF rtHomingCancel.Q THEN
	bHomingDone							:= FALSE;

END_IF

//Jeśli na wejsciu pojawi sie ustawianie aktualnej pozycji enkodera
rtActuatorPositionSet(CLK:=bPositionSet,Q=>);
IF rtActuatorPositionSet.Q THEN
	bEncoderReset						:= TRUE;
	nEncoderResetVal					:= 0;
	bHomingDone							:= TRUE;
;
END_IF

IF bEncoderSetDone THEN
	bEncoderReset						:= FALSE;
END_IF

////Zapisywanie ostatniego kierunku ruchu siłownika
//IF bUpDirectionOut AND NOT bDownDirectionOut THEN
//	bLastDirectionUp:=TRUE;
//ELSIF bDownDirectionOut AND NOT bUpDirectionOut THEN
//	bLastDirectionUp:=FALSE;	
//END_IF

////Wykrywanie zbocza pulsu enkodera
//rtEncoderPulse(CLK:=bEncoderPulse,Q=>);
//ftEncoderPulse(CLK:=bEncoderPulse,Q=>);

//tonOffDelay(IN:= NOT bUpDirectionOut AND NOT bDownDirectionOut, PT:=T#2S);

//IF NOT bOptionCoutingFalling THEN
//	IF rtEncoderPulse.Q OR ftEncoderPulse.Q THEN
//		IF bLastDirectionUp THEN
//			lrActuatorPosition:=lrActuatorPosition+rPulseRatio;
//		ELSE
//			lrActuatorPosition:=lrActuatorPosition-rPulseRatio;
//		END_IF	
//	END_IF
//ELSE
//	IF (bUpDirectionOut OR bDownDirectionOut) THEN
//		IF rtEncoderPulse.Q OR ftEncoderPulse.Q THEN
//			IF bLastDirectionUp THEN
//				lrActuatorPosition:=lrActuatorPosition+rPulseRatio;
//			ELSE
//				lrActuatorPosition:=lrActuatorPosition-rPulseRatio;
//			END_IF	
//		END_IF
//	ELSIF (NOT tonOffDelay.Q AND (rtEncoderPulse.Q OR ftEncoderPulse.Q)) THEN
//		lrActuatorPosition:=lrActuatorPosition-rPulseRatio;
//		cnt:=cnt +1;
//	END_IF	
//END_IF

END_FUNCTION_BLOCK

// ---- POUs/FB/NewFBs/FB_FormsDragStepper.TcPOU
(*
Nazwa:		FB_FormsDragStepper
Opis:		Przeciąganie formatek 
Wersja:		V0.22
Data:		2025-09-04
Autor:		DJ, DP
Urządzenia:	Siłownik podnoszenia wideł, Silnik krokowy przeciągania 
Ostatnie zmiany:
	- 20250904 [DP] EventLog->wywołać błędy 
	- 2025-08-19 [DP] Homing false
	- 2024-11-25 [DP] Czujnik dół
	- 2024-10-01 [DP] ESTOP Delay
	- RRRR-MM-DD [KTO?] Tekst Tekst Tekst Tekst Tekst Tekst Tekst Tekst Tekst Tekst 
	- 2025-09-15[VS] Jazda i stop w pozycji końcowej
Konfiguracja:
	- Krokówka
	Instukcja:
		-
		-
		-
	
Info:
	- Obsługa tylko jednego siłownika podnoszenia i dwóch siłowników prowadzących

*)

FUNCTION_BLOCK FB_FormsDragStepper
VAR_INPUT
	bEnable										: BOOL;				//Zezwolenie na pracę
	bEStop										: BOOL;				//Stop awaryjny włączony
	bRun										: BOOL;				//Rozkaz przeciagania
	bPrepare									: BOOL;				//Rozkaz przygotownaia 
	bDragUpWhenReady							: BOOL;					
	bHoming										: BOOL;				//Zezwolenie na wykonanie bazowania i pozycjonowanie układu
	bHomingDirection							: BOOL;				//Kierunek bazowania
	bBefore2ActuatorOff							: BOOL;
	bDelayAfterDrag								: BOOL;				//Opóżnienie po przeciąganiu
	bHeightSet									: BOOL;				//Ustaw do pozycji
	bIgnoreError								: BOOL;				//Ignorowanie błędów 
	bReset										: BOOL;				//Reset błędu, jeśli jest w stanie "eError"
	bResetCycle									: BOOL;				//Reset cyklu

	bTwoPhaseMode								: BOOL;				//Załączone dozowanie dwufazowe
	lrMinPosition								: LREAL;			 	
	lrMaxPosition								: LREAL;			 		
	lrStartPosition								: LREAL;			//Zadane położenie 
	lrMiddlePosition							: LREAL;			//Zadane położenie 
	lrEndPosition								: LREAL;			//Zadane położenie 		
	lrStartPositionTwoPhase						: LREAL;			//Zadane położenie 
	lrMiddlePositionTwoPhase					: LREAL;			//Zadane położenie 
	lrEndPositionTwoPhase						: LREAL;			//Zadane położenie 	
	lrLeadActuatorMoveUpPosition				: LREAL;			//Zadane położenie 	
	lrDragAcceleration							: LREAL;			//Przyspieszenie 
	lrDragDeceleration							: LREAL;			//Opóźnienie 
	lrDragJerk									: LREAL;			//Jerk
	lrDragSpeed									: LREAL;			//Prędkość 
	
	bHomingSensor								: BOOL;				//Czujnik bazowania 
	bDragUpSensor								: BOOL;				//
	bDragDownSensor								: BOOL;				//
	bLead1UpSensor								: BOOL;				//
	bLead2UpSensor								: BOOL;				//
	bManualMovement								: BOOL;				//Zezwolenie na ruchy ręczne

	_ALARMINFO_									: BOOL;
	iStationIndex								: UDINT;
	wsStationName								: WSTRING;
	bMoveToEndPosition							: BOOL;					//ustawienie w końcowej pozycji dla uruchomienia
END_VAR

VAR_OUTPUT
	eState										: E_Station;
	eRunningState								: E_DragStationState;	// Stan przeciągania formatek
	bError										: BOOL;					// Błąd stacji
	udiErrorID									: UDINT;				// Nr blędu przeciągania formatek
	sErrorDescription							: STRING(200);			// Opis błędu
	sErrorDescription2							: STRING(200);			// Opis błędu
	sErrorStationName							: STRING;				// Nazwa stacji
	udiStationID								: UDINT;				// Nr stacji

	bDragActuator								: BOOL;					
	bLeadBefore1Actuator						: BOOL;					
	bLeadBefore2Actuator						: BOOL;					
	
	bCycleDone									: BOOL;					//Sygnał zakończenia cyklu
	bCycleNotDone								: BOOL;
	bHomingDone									: BOOL;
	tCycleTime									: TIME;					//Czas cyklu
	lrActualDragPosition						: LREAL;				//Aktualne położenie
	//Dodatkowe	
	eRunningStateBeforeEStop					: E_DragStationState;	//Stan przed E-Stopem	
	bWasErrorOrEstop							: BOOL;
	
END_VAR

VAR
	(*LastStates*)
	eLastState									: E_Station;						//Stan ogólny bloku
	eLastStateTemp								: E_Station;						//Stan ogólny bloku
	eLastRunningState							: E_DragStationState;				//Stan podbloku
	eLastRunningStateTemp						: E_DragStationState;				//Stan podbloku
	
	(*Axis online*)
	fbDrag										: FB_McAxisOnlineNC;
	stDrag										: ST_McAxisOnline;
	                                    		                                 		
	(*Control*)
	tonResetting								: TON;								//Czas resetu
	tonHoming									: TON;
	tonPreparingToReady							: TON;								//Czas potrzeby na przygotowanie osi
	rtResetCommands								: R_TRIG;                                    	
	rtResetCycle								: R_TRIG;

	(*Statistics*)
	tonCycleTimer								: TON;								//Czas cyklu przeciągania	
	rtrigCycleTimerRead							: R_TRIG;

	(*Homing*)
	iHomingCase									: INT;
	
	(*Aborting*)
	iAbortingCase								: INT;
	                                    	
	(*Errors*)
	bStateError									: BOOL;
	tonEstopDelay								: TON;
	bResetCycleOn								: BOOL;
	tonbDragUpSensor							: TON;	
	tonbDragDownSensor							: TON;		
	tonbLead1UpSensor							: TON;
	tonbLead2UpSensor							: TON;
	
	(*Running*)

	tonNotDragActuatorDelay						: TON;
	tonRunningDraging							: TON;
	tonRunningeEndingOfDrag						: TON;
	(*Inne*)
	
		//Zmienne od EVENTLOGGER
	bAlarmInit 						: BOOL := TRUE; 
	nAlarmNumerator					: INT;
	arfbAlarm						: ARRAY[0..19] OF  FB_TcAlarm;		//Tablica bloczków błędów
	fbSourceInfo 					: FB_TcSourceInfo;
	iSourceInfo						: I_TcSourceInfo;
	sAlarmTest						: STRING;
	//Koniec zmiennych od EVENTLOGGER
	
END_VAR
	
VAR_IN_OUT
	bManualDragActuator							: BOOL;		
	bManualLeadBefore1Actuator					: BOOL;			
	bManualLeadBefore2Actuator					: BOOL;			
	bManualDragRight							: BOOL;				
	bManualDragLeft								: BOOL;		
	DragAxisRef									: AXIS_REF;		
END_VAR

ResetAll();
ErrorHandling();
Signals();
Control();
Limits();
DragControlBlocks();
Statistics();
aStationID();
(*Zapisywanie ostatniego stanu*)
IF eLastStateTemp<>eState THEN
	eLastState := eLastStateTemp;
END_IF
eLastStateTemp := eState;
IF eLastRunningStateTemp<>eRunningState THEN
	eLastRunningState := eLastRunningStateTemp;
END_IF
eLastRunningStateTemp := eRunningState;
(*Koniec Zapisywanie ostatniego stanu*)

ACTION aStationID:
udiStationID	:=	iStationIndex;
END_ACTION

ACTION Control:


	(*****Wyłączenie enable*****)
	IF NOT bEnable AND NOT bError THEN
		IF eState <> E_Station.eDisabled AND eState <> E_Station.ePreparingToDisable THEN
				eState 								:= E_Station.ePreparingToDisable; 
		END_IF	
	END_IF

	(*****Estop*****)
	IF NOT bEstop  THEN	
		IF eState <> E_Station.eAborted AND eState <> E_Station.eAborting AND eState <> E_Station.eDisabled THEN
				eRunningStateBeforeEStop			:= eRunningState;
				eState 								:= E_Station.eAborting; 
				iAbortingCase						:= 0; 
		END_IF
	END_IF


	
CASE eState OF
	
//==========================================================================================	
	E_Station.eDisabled: 						// Stan nieaktywnosci (Stacja wyłączona) 
		
		IF bEnable THEN
			eState 									:= E_Station.ePreparingToReady; 
		END_IF 

//==========================================================================================	    
	E_Station.eAborted: 						// Stan bezpiecznego zatrzymania (po Abortingu) 	
			
		IF bEStop THEN
			bWasErrorOrEstop						:= TRUE;	
			eState 									:= E_Station.ePreparingToReady;
		END_IF		
			
//==========================================================================================	
	E_Station.eAborting:                 		// Stan bezpiecznego zatrzymywania (po EStopie)
		
		CASE iAbortingCase OF
			
			0: //Inicjalizacja
				IF stDrag.mcPower.bStatus THEN
					iAbortingCase					:= 10;
				ELSE
					iAbortingCase					:= 40;
				END_IF
				
			10: //Komenda MC_STOP
				stDrag.mcStop.bExecute				:= TRUE;	
				//Czekam na Done
				IF stDrag.mcStop.bDone THEN
					stDrag.mcStop.bExecute			:= FALSE;
					iAbortingCase					:= 20;
				END_IF
				
			20: //Kasowanie komend
				stDrag.mcMoveAbsolute.bExecute		:= FALSE;
				stDrag.mcMoveRelative.bExecute		:= FALSE;
				ResetCommands();
				iAbortingCase						:= 30;
	
			30: //Wyłączenie osi
				stDrag.mcPower.bEnable				:= FALSE;
				stDrag.mcPower.bEnable_Negative		:= FALSE;
				stDrag.mcPower.bEnable_Positive		:= FALSE;
				IF NOT stDrag.mcPower.bStatus THEN
					iAbortingCase					:= 40;
				END_IF
				
			40: //Kasowanie podzespołow
				ResetCommands();
				iAbortingCase						:= 50;
				
			50: //Przejście do Aborted
				iAbortingCase						:= 0;
				eState								:= E_Station.eAborted;
				eRunningState						:= E_DragStationState.eReady;
				
		END_CASE

//==========================================================================================			
	E_Station.eError:                 	 		// Stan błędu 	
		
		bWasErrorOrEstop							:= TRUE;

		IF bReset THEN
			eState									:= E_Station.eResetting;	
		ELSE
			ResetCommands();
		END_IF
			
//==========================================================================================
	E_Station.eResetting:						// Stan resetowania bledu (po Errorze)
			
	//Procedura obsługi resetu w zależności od błędu
//	CASE udiErrorID OF 
//	CASE udiErrorID - iStationIndex(*udiResetStep*) OF 	
//		171: //Error 1 - Błąd Serwa
		IF  arfbAlarm[0].bActive THEN
			stDrag.mcReset.bExecute					:= TRUE;
			IF stDrag.mcReset.bDone THEN
				stDrag.mcReset.bExecute				:= FALSE;
				bError								:= FALSE;
			END_IF	
		END_IF
		
//		172,173://Error 2 - Błąd siłownika przeciągania
		IF  arfbAlarm[1].bActive OR arfbAlarm[2].bActive THEN
			bDragActuator							:= FALSE;	
			//bLeadBefore1Actuator					:= FALSE;				
			//bLeadBefore2Actuator					:= FALSE;			
			bError									:= FALSE;
		END_IF	
// 		174: //Error 4 - Błąd siłownika prowadzenia
		IF arfbAlarm[3].bActive THEN
			//bDragActuator							:= FALSE;	
			bLeadBefore1Actuator					:= TRUE;				
			//bLeadBefore2Actuator					:= FALSE;			
			bError									:= FALSE;		
		END_IF
// 		175: //Error 5 - Błąd siłownika prowadzenia
		IF arfbAlarm[4].bActive THEN
			//bDragActuator							:= FALSE;	
			bLeadBefore2Actuator					:= NOT bBefore2ActuatorOff;				
			//bLeadBefore2Actuator					:= FALSE;			
			bError									:= FALSE;		
		END_IF
//	END_CASE
	
	IF NOT bError THEN
		udiErrorID									:= 0;
		sErrorDescription							:= '';
		sErrorDescription2							:= '';	
		eState										:= E_Station.ePreparingToReady;
	ELSIF tonResetting.Q THEN                   	
		eState										:= E_Station.eError;
	END_IF	
 
//==========================================================================================
	E_Station.eManualMovement:     				// Stan ruchów manualnych  
       
		ManualMovements();
		//Wyjście z trybu serwisowego
		IF NOT bManualMovement THEN
			bDragActuator							:=	bManualDragActuator;	
			bLeadBefore1Actuator					:=	bManualLeadBefore1Actuator;
			bLeadBefore2Actuator					:=	bManualLeadBefore2Actuator;
			eState									:=	E_Station.eReady;
		END_IF 

//==========================================================================================		
	E_Station.eHoming:							// Stan bazowania 
		
		Homing();	
		IF NOT bHoming AND NOT bHeightSet AND tonHoming.Q THEN
			eState									:=	E_Station.ePreparingToReady;
		END_IF		
			
//==========================================================================================
	E_Station.eHomingDone:                  	// Stan wykonania bazowania 

		bHomingDone									:= TRUE;
		bResetCycleOn								:= FALSE;		
		IF NOT bHoming AND NOT bHeightSet AND NOT bResetCycleOn THEN
		//	eState									:=	E_Station.eReady;
			eState									:=	E_Station.ePreparingToReady;
		END_IF

//==========================================================================================
	E_Station.ePreparingToReady:            	// Stan przygotowywania do gotowosci (zawsze przed Ready)  

		IF tonPreparingToReady.Q THEN
			
			stDrag.mcPower.bEnable					:= TRUE;
			stDrag.mcPower.bEnable_Negative			:= TRUE;
			stDrag.mcPower.bEnable_Positive			:= TRUE;
			stDrag.mcPower.lrOverride				:= 100;
			
			IF stDrag.mcPower.bStatus THEN
				
				ResetCommands();
				eState								:= E_Station.eReady;
				eRunningState						:= E_DragStationState.eReady;
				
				IF bResetCycleOn THEN
					eState							:= E_Station.eHoming;
				END_IF
				
			END_IF
		
		END_IF			

//==========================================================================================
	E_Station.ePreparingToDisable:         	 	// Stan przygotowywania do nieaktywnosci (po wyłączeniu Enable) 
  
		stDrag.mcPower.bEnable						:= FALSE;
		stDrag.mcPower.bEnable_Negative				:= FALSE;
		stDrag.mcPower.bEnable_Positive				:= FALSE;
		stDrag.mcPower.lrOverride					:= 0;
		
		bWasErrorOrEstop							:= FALSE;
		bHomingDone									:= FALSE;	
		
		IF NOT stDrag.mcPower.bStatus THEN
			ResetCommands();
			eState									:= 	E_Station.eDisabled;
			eRunningState							:= 	E_DragStationState.eReady;
		END_IF

//==========================================================================================	
	E_Station.eReady:							// Stan gotowosci 


		(*Skasowanie wszystkich komend*)
		IF rtResetCommands.Q THEN	ResetCommands();	END_IF		
		
		IF bDragUpWhenReady THEN
			bDragActuator							:=	TRUE;
		END_IF
	
		IF (bRun OR bPrepare) AND NOT bCycleDone THEN
			eState									:= E_Station.eStarting;
			//IF bDragUpWhenReady THEN
				bDragActuator						:=	FALSE;
			//END_IF			
		END_IF		
		IF bHoming OR bHeightSet THEN
			eState									:= E_Station.eHoming;
		END_IF
		IF bManualMovement THEN
			bManualDragActuator						:=	bDragActuator;			
			bManualLeadBefore1Actuator				:=	bLeadBefore1Actuator;	
			bManualLeadBefore2Actuator				:=	bLeadBefore2Actuator;	
			bManualDragRight						:=	FALSE;		
			bManualDragLeft							:=	FALSE;					
			eState									:= E_Station.eManualMovement;					
		END_IF
		IF NOT bRun AND NOT bPrepare THEN
			bCycleDone								:= FALSE;
		END_IF

//==========================================================================================
	E_Station.eStopping:					// Stan zatrzymywania 
		
		Running();
		
		//Czekam dopóki skończy ruch
		IF	eRunningState <> E_DragStationState.eDraging AND eRunningState <> E_DragStationState.eDragingDone AND eRunningState <> E_DragStationState.eEndingOfDrag AND eRunningState <> E_DragStationState.eDraged
		AND  eRunningState <> E_DragStationState.eEndingOfDragDone AND  eRunningState <> E_DragStationState.eLowering  THEN	
			stDrag.mcReset.bExecute					:= TRUE;	
		END_IF
		
		//Reset ruchu
		IF stDrag.mcReset.bDone THEN		
			stDrag.mcReset.bExecute					:= FALSE;
			eState 									:= E_Station.eReady;
		END_IF

//==========================================================================================
	E_Station.eStarting:                  	// Stan uruchamiania (po Ready)
		
		eState										:= E_Station.eRunning;

//==========================================================================================
	E_Station.eRunning:               		// Stan wykonywania cyklu (po Startingu), w tym stanie osobny
 
		Running();

		IF NOT bRun AND NOT bPrepare THEN					(*Przerywanie cyklu*)
			eState 				 					:= E_Station.eStopping;	
		END_IF
			
		IF bCycleDone THEN (*Cykl zakończony*)
			eState 				 					:= E_Station.eReady;
		END_IF	
		
//==========================================================================================
END_CASE
END_ACTION

ACTION DragControlBlocks:
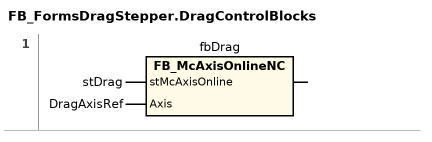
// NETWORK 1
fbDrag(stMcAxisOnline := stDrag, Axis := DragAxisRef); // FB_McAxisOnlineNC
END_ACTION

ACTION ErrorHandling:
// Alarm_0260	260	Error	Błąd napędu przeciągania. Błąd NC: {0}
// Alarm_0261	261	Error	Siłownik przeciągania | Blokada podnoszenia - sprawdź czujnik lub odblokuj
// Alarm_0262	262	Error	Siłownik przeciągania | Blokada opuszczania siłownika - sprawdź czujnik lub odblokuj
// Alarm_0263	263	Error	Siłownik prowadzenia | Blokada podnoszenia - sprawdź czujnik lub odblokuj
// Alarm_0264	264	Error	Siłownik prowadzenia | Blokada podnoszenia - sprawdź czujnik lub odblokuj

IF bAlarmInit THEN
    bAlarmInit := FALSE; 
	fbSourceInfo.Clear();
	fbSourceInfo.sName:=wsLiteral_TO_UTF8(wsStationName);//'Machine';
	fbSourceInfo.nId:=iStationIndex;//2700;
	// Alarm_0260	260	Error	Błąd napędu przeciągania. Błąd NC: {0}
    arfbAlarm[0].CreateEx(stEventEntry := TC_EVENTS.AlarmClass.Alarm_0260, bWithConfirmation:= FALSE,  ipSourceInfo:= fbSourceInfo); 
	// Alarm_0261	261	Error	Siłownik przeciągania | Blokada podnoszenia - sprawdź czujnik lub odblokuj
	arfbAlarm[1].CreateEx(stEventEntry := TC_EVENTS.AlarmClass.Alarm_0261, bWithConfirmation:= FALSE,  ipSourceInfo:= fbSourceInfo);
	// Alarm_0262	262	Error	Siłownik przeciągania | Blokada opuszczania siłownika - sprawdź czujnik lub odblokuj
	arfbAlarm[2].CreateEx(stEventEntry := TC_EVENTS.AlarmClass.Alarm_0262, bWithConfirmation:= FALSE,  ipSourceInfo:= fbSourceInfo);
	// Alarm_0263	263	Error	Siłownik prowadzenia | Blokada podnoszenia - sprawdź czujnik lub odblokuj
	arfbAlarm[3].CreateEx(stEventEntry := TC_EVENTS.AlarmClass.Alarm_0263, bWithConfirmation:= FALSE,  ipSourceInfo:= fbSourceInfo);
	// Alarm_0264	264	Error	Siłownik prowadzenia | Blokada podnoszenia - sprawdź czujnik lub odblokuj
	arfbAlarm[4].CreateEx(stEventEntry := TC_EVENTS.AlarmClass.Alarm_0264, bWithConfirmation:= FALSE,  ipSourceInfo:= fbSourceInfo);

	
END_IF

//CZYTANIE STATUSÓW
DragAxisRef.ReadStatus();

bStateError										:= (eState=E_Station.eError) OR (eState=E_Station.eResetting) OR NOT bEstop OR bIgnoreError;
tonEstopDelay									(IN:=bEStop,	PT:=T#4S);

IF bEnable AND tonEstopDelay.Q THEN
	// Alarm_0260	260	Error	Błąd napędu przeciągania. Błąd NC: {0}
	//Error 1 - Błąd Serwa
	IF stDrag.bError THEN
		bHomingDone									:= FALSE;	
		arfbAlarm[0].ipArguments.Clear() .AddString(stDrag.stError.sNcError);
		IF NOT arfbAlarm[0].bActive THEN
			stDrag.mcReset.bExecute				:= TRUE; // na testy jak wystąpi błąd
			arfbAlarm[0].Raise(nTimeStamp:=0);
		END_IF
	ELSE	
		IF  arfbAlarm[0].bActive AND bReset THEN
			arfbAlarm[0].Clear(nTimeStamp:=0, bResetConfirmation:= FALSE);
		END_IF	
// 		stDrag.mcReset.bExecute				:= TRUE; // na testy jak wystąpi błąd
// 		bError								:= TRUE;
// 		udiErrorID							:= 171;
// 		//udiErrorID							:= udiErrorID + iStationIndex;
// 		sErrorDescription					:= 'Błąd napędu przeciągania. Błąd NC:';
// 		sErrorDescription2					:= stDrag.stError.sNcError;
	END_IF
	
	//Alarm_0261	261	Error	Siłownik przeciągania | Blokada podnoszenia - sprawdź czujnik lub odblokuj
	//Error 2 - Błąd siłownika przeciągania
	tonbDragUpSensor	(IN:= bDragActuator AND NOT bDragUpSensor	, PT:=T#2S);
	IF tonbDragUpSensor.Q THEN
		bHomingDone									:= FALSE;			
		IF NOT arfbAlarm[1].bActive THEN
			arfbAlarm[1].Raise(nTimeStamp:=0);
		END_IF
	ELSE	
		IF  arfbAlarm[1].bActive AND bReset THEN
			arfbAlarm[1].Clear(nTimeStamp:=0, bResetConfirmation:= FALSE);
		END_IF	
// 		bError								:= TRUE;
// 		udiErrorID							:= 172;	
// 		//udiErrorID 							:= udiErrorID + iStationIndex;
// 		sErrorDescription					:= 'Siłownik przeciągania';
// 		sErrorDescription2					:= 'Blokada podnoszenia - sprawdź czujnik lub odblokuj';
	END_IF
	
	// Alarm_0262	262	Error	Siłownik przeciągania | Blokada opuszczania siłownika - sprawdź czujnik lub odblokuj
	//Error 3 - Błąd siłownika przeciągania
	tonbDragDownSensor	(IN:= NOT bDragActuator AND NOT bDragDownSensor	AND bRun, PT:=T#2S);
	IF tonbDragDownSensor.Q THEN
		IF NOT arfbAlarm[2].bActive THEN
			arfbAlarm[2].Raise(nTimeStamp:=0);
		END_IF
	ELSE	
		IF  arfbAlarm[2].bActive AND bReset THEN
			arfbAlarm[2].Clear(nTimeStamp:=0, bResetConfirmation:= FALSE);
		END_IF	
// 		bError								:= TRUE;
// 		udiErrorID							:= 173;	
// 		//udiErrorID 							:= udiErrorID + iStationIndex;
// 		sErrorDescription					:= 'Siłownik przeciągania';
// 		sErrorDescription2					:= 'Blokada opuszczania siłownika - sprawdź czujnik lub odblokuj';
	END_IF;			
	
	// Alarm_0263	263	Error	Siłownik prowadzenia | Blokada podnoszenia - sprawdź czujnik lub odblokuj
	//Error 4 - Błąd siłownika prowadzenia
	tonbLead1UpSensor	(IN:= bLeadBefore1Actuator AND NOT bLead1UpSensor	, PT:=T#2S);
	IF tonbLead1UpSensor.Q THEN
		IF NOT arfbAlarm[3].bActive THEN
			arfbAlarm[3].Raise(nTimeStamp:=0);
		END_IF
	ELSE	
		IF  arfbAlarm[3].bActive AND bReset THEN
			arfbAlarm[3].Clear(nTimeStamp:=0, bResetConfirmation:= FALSE);
		END_IF	
// 		bError								:= TRUE;
// 		udiErrorID							:= 174;	
// 		//udiErrorID 							:= udiErrorID + iStationIndex;
// 		sErrorDescription					:= 'Siłownik prowadzenia';
// 		sErrorDescription2					:= 'Blokada podnoszenia - sprawdź czujnik lub odblokuj';
	END_IF;		
	
	//// Alarm_0264	264	Error	Siłownik prowadzenia | Blokada podnoszenia - sprawdź czujnik lub odblokuj
	//Error 5 - Błąd siłownika prowadzenia
	tonbLead2UpSensor	(IN:= bLeadBefore2Actuator AND NOT bLead2UpSensor	, PT:=T#2S);
	IF tonbLead2UpSensor.Q THEN
		IF NOT arfbAlarm[4].bActive THEN
			arfbAlarm[4].Raise(nTimeStamp:=0);
		END_IF
	ELSE	
		IF  arfbAlarm[4].bActive AND bReset THEN
			arfbAlarm[4].Clear(nTimeStamp:=0, bResetConfirmation:= FALSE);
		END_IF	
// 		bError								:= TRUE;
// 		udiErrorID							:= 175;	
// 		//udiErrorID 							:= udiErrorID + iStationIndex;
// 		sErrorDescription					:= 'Siłownik prowadzenia';
// 		sErrorDescription2					:= 'Blokada podnoszenia - sprawdź czujnik lub odblokuj';
	END_IF;		
ELSE
	bError := FALSE;
END_IF

//******************PRZEJŚCIE DO eERROR*****************************

IF bError AND  NOT bStateError THEN
	eState 									:= E_Station.eError;
END_IF

//****************WYŚWIETLANIE STATUSU BLEDU************************
(*Wyświetlanie błedu na wyjściu*)
bError							:= FALSE;
FOR nAlarmNumerator := 0 TO 19 DO
	bError						:= bError OR arfbAlarm[nAlarmNumerator].bActive;
END_FOR

(*Przepisywanie nazwy stacji*)
sErrorStationName 							:= WSTRING_TO_STRING(wsStationName);
END_ACTION

ACTION Homing:

stDrag.mcMoveRelative.lrAcceleration			:=	1500;
stDrag.mcMoveRelative.lrDeceleration			:=	1500;
stDrag.mcMoveRelative.lrJerk					:=	15000;
stDrag.mcMoveRelative.lrVelocity				:=	15;

stDrag.mcMoveVelocity.lrAcceleration			:= 	2500;
stDrag.mcMoveVelocity.lrDeceleration			:= 	2500;
stDrag.mcMoveVelocity.lrJerk					:= 	2500;
stDrag.mcMoveVelocity.lrVelocity				:= 	10;	

stDrag.stStatus.lrPosDiff;
stdrag.stStatus.lrActPos;

IF bHoming THEN // Bazowanie - podjazd do góry i ustawienie obrotu
	CASE iHomingCase OF
	
	0: //Opuszczamy widły
		bHomingDone										:= FALSE;
		                                        		
		stDrag.mcMoveAbsolute.bExecute					:= FALSE;
		stDrag.mcMoveRelative.bExecute					:= FALSE;
		stDrag.mcMoveVelocity.bExecute					:= FALSE;
		
		bDragActuator									:= FALSE;	
		bLeadBefore1Actuator							:= TRUE; 	
		bLeadBefore2Actuator							:= NOT bBefore2ActuatorOff;
			
		iHomingCase										:= 10;
	
	10: //Sprawdzamy czy jest na czujniku
		IF bHomingSensor THEN
			iHomingCase									:= 20;
		ELSE                                        	
			iHomingCase									:= 30;
		END_IF
		
	20: //Muszę wyjechać z czujnika
		stDrag.mcMoveRelative.lrAcceleration			:=1500;
		stDrag.mcMoveRelative.lrDeceleration			:=1500;
		stDrag.mcMoveRelative.lrJerk					:=15000;
		stDrag.mcMoveRelative.lrVelocity				:=15;

		stDrag.mcMoveRelative.lrDistance				:= 50; // bylo 50
		IF bHomingDirection THEN
			stDrag.mcMoveRelative.lrDistance			:= -50; // bylo 50
		END_IF
		
		stDrag.mcMoveRelative.bExecute					:= TRUE;
		
		IF stDrag.mcMoveRelative.bDone THEN
			stDrag.mcMoveRelative.bExecute				:= FALSE;
			iHomingCase									:= 30;
		END_IF
		
	30: //Bazuje na czujnik
		stDrag.mcMoveVelocity.lrAcceleration			:= 2500;
		stDrag.mcMoveVelocity.lrDeceleration			:= 2500;
		stDrag.mcMoveVelocity.lrJerk					:= 2500;
		stDrag.mcMoveVelocity.lrVelocity				:= 10;	
	
		stDrag.mcMoveVelocity.eDirection				:= MC_Negative_Direction;
		IF bHomingDirection THEN
			stDrag.mcMoveVelocity.eDirection			:= MC_Positive_Direction;
		END_IF
		
		stDrag.mcMoveVelocity.bExecute					:= TRUE;
		
		IF bHomingSensor THEN
			stDrag.mcMoveVelocity.bExecute				:= FALSE;
			iHomingCase									:= 40;
		END_IF
		
	40: //Zatrzymanie osi
		stDrag.mcStop.bExecute							:= TRUE;
		
		IF stDrag.mcStop.bDone THEN
			stDrag.mcStop.bExecute						:= FALSE;
			iHomingCase									:= 50;
		END_IF
	
	50: 

		iHomingCase										:= 60;
		
	60: //Bazujemy Enkoder
		stDrag.mcHome.eHomingMode						:= MC_Direct;
		stDrag.mcHome.lrPosition						:= lrMinPosition;
		IF bHomingDirection THEN
			stDrag.mcHome.lrPosition					:= lrMaxPosition;
		END_IF
		
		stDrag.mcHome.bExecute							:= TRUE;
		                                        		
		IF stDrag.mcHome.bDone THEN             		
			stDrag.mcHome.bExecute						:= FALSE;
			iHomingCase									:= 70;
		END_IF
		
	70:                             	
		iHomingCase										:= 80;

	80:
		stDrag.mcMoveAbsolute.lrAcceleration			:=1500;
		stDrag.mcMoveAbsolute.lrDeceleration			:=1500;
		stDrag.mcMoveAbsolute.lrJerk					:=15000;
		stDrag.mcMoveAbsolute.lrVelocity				:=15;
									  
		stDrag.mcMoveAbsolute.lrPosition			  	:= lrStartPosition;
		stDrag.mcMoveAbsolute.bExecute				  	:= TRUE;
			
		IF stDrag.mcMoveAbsolute.bDone THEN
			stDrag.mcMoveAbsolute.bExecute				:= FALSE;
			iHomingCase									:= 100;
		END_IF	
		
	100: //Zbazowano	
		iHomingCase										:= 0;
		eState											:= E_Station.eHomingDone;
	
	END_CASE
END_IF	
IF bHeightSet THEN

	bDragActuator									:= FALSE;	
	bLeadBefore1Actuator							:= FALSE;	
	bLeadBefore2Actuator							:= FALSE;

	//Dynamika Ruchu
	stDrag.mcMoveAbsolute.lrAcceleration			:= lrDragAcceleration;
	stDrag.mcMoveAbsolute.lrDeceleration			:= lrDragDeceleration;
	stDrag.mcMoveAbsolute.lrVelocity				:= lrDragSpeed;
	stDrag.mcMoveAbsolute.lrJerk					:= 10000;
	                                            	                     	
	stDrag.mcMoveAbsolute.lrPosition				:= lrStartPosition;                                            	
	stDrag.mcMoveAbsolute.bExecute					:= TRUE;
	                                            	
	IF stDrag.mcMoveAbsolute.bDone THEN         	
		stDrag.mcMoveAbsolute.bExecute				:= FALSE;
		eState										:= E_Station.eHomingDone;
	END_IF
		
END_IF
END_ACTION

ACTION Limits:
(*Wywowyłanie na początku*)


(*Prędkość zakręcania*)


(*Inny parametr*)
//...
END_ACTION

ACTION ManualMovements:

IF NOT bRun AND NOT bPrepare AND bManualMovement THEN
	stDrag.mcJog.bJogForward						:=	bManualDragRight AND	lrActualDragPosition < lrEndPosition AND NOT bLeadBefore1Actuator;
	stDrag.mcJog.bJogBackwards						:=	bManualDragLeft AND		lrActualDragPosition > lrStartPosition AND NOT bLeadBefore1Actuator;                                  	                                  	                                   	
	bDragActuator									:=	bManualDragActuator;			
	bLeadBefore1Actuator							:=	bManualLeadBefore1Actuator;	
	bLeadBefore2Actuator							:=	bManualLeadBefore2Actuator;	
ELSE
	bManualDragActuator								:=	FALSE;		
	bManualLeadBefore1Actuator						:=	FALSE;		
	bManualLeadBefore2Actuator						:=	FALSE;		
END_IF
	
IF bHoming OR bHeightSet THEN
	eState											:=	E_Station.eHoming;	
END_IF                                                	

IF  (bRun OR bPrepare) AND bManualMovement THEN                                                     	
	Running();
END_IF

IF NOT bRun AND NOT bPrepare THEN
	bCycleDone 										:= FALSE;
	bCycleNotDone 									:= FALSE;	
END_IF
END_ACTION

ACTION ResetAll:
(*****Reset bloczka*****)
IF bEnable THEN
	IF eState <> E_Station.eDisabled AND eState <> E_Station.ePreparingToDisable THEN
		IF bResetCycle THEN
			bResetCycleOn						:= TRUE;
			eState								:= E_Station.ePreparingToReady;
		END_IF
	END_IF
END_IF


IF bResetCycleOn THEN
	
	ResetCommands();
	eRunningState							:= E_DragStationState.eReady;	
	eState 				 					:= E_Station.eReady;

END_IF
END_ACTION

ACTION ResetCommands:
//KAsowanie komend ruchu 
stDrag.mcJog.bJogForward								:=	FALSE;
stDrag.mcJog.bJogBackwards								:=	FALSE;
stDrag.mcHome.bExecute									:=	FALSE;
                                                          	
stDrag.mcMoveAbsolute.bExecute							:=	FALSE;
stDrag.mcMoveRelative.bExecute							:=	FALSE;
stDrag.mcMoveVelocity.bExecute							:=	FALSE;
                                                          	
stDrag.mcStop.bExecute									:=	FALSE;
stDrag.mcReset.bExecute									:=	FALSE;
                                                          	
bManualDragActuator										:=	FALSE;		
bManualLeadBefore1Actuator								:=	FALSE;	
bManualLeadBefore2Actuator								:=	FALSE;	
bManualDragRight										:=	FALSE;	
bManualDragLeft											:=	FALSE;	
                                                          	
bDragActuator											:=	FALSE;	
bLeadBefore1Actuator									:=	TRUE;	
bLeadBefore2Actuator									:=	NOT bBefore2ActuatorOff;
                                                          	
bResetCycleOn											:=	FALSE;	

iHomingCase												:=	0;
//bCycleDone								   				:=	FALSE;
END_ACTION

ACTION Running:
	
CASE eRunningState OF
	
	E_DragStationState.eDisabled:
		eRunningState								:= E_DragStationState.eReady; 
	
	E_DragStationState.eReady:
		IF NOT bMoveToEndPosition THEN
			IF NOT bCycleDone  THEN                                           	
				IF bRun OR bPrepare THEN   
					bDragActuator								:=	FALSE;
					eRunningState								:=	E_DragStationState.ePreparingToMove; 
       			END_IF
			END_IF
		ELSE
			bDragActuator								:=	TRUE;
			bLeadBefore1Actuator						:=	TRUE;
			bLeadBefore2Actuator						:=	TRUE;
			IF bRun OR bPrepare THEN   
					eRunningState								:=	E_DragStationState.ePreparingToMove; 
       			END_IF
		END_IF	
		//Po E-Stopie
(*		IF bWasErrorOrEstop THEN	
			bWasErrorOrEstop						:= FALSE;
			eRunningState							:= eRunningStateBeforeEStop;
		END_IF*)
		
// Sygnal przygotowania do przeciaganiecia formatek		
	E_DragStationState.ePreparingToMove:
	
		stDrag.mcMoveAbsolute.lrAcceleration		:= lrDragAcceleration;
		stDrag.mcMoveAbsolute.lrDeceleration		:= lrDragDeceleration;
		stDrag.mcMoveAbsolute.lrJerk				:= lrDragJerk;
		stDrag.mcMoveAbsolute.lrVelocity			:= lrDragSpeed;

		IF NOT bMoveToEndPosition THEN
			stDrag.mcMoveAbsolute.lrPosition			:= lrStartPosition;
			IF bTwoPhaseMode THEN //dwu-faza
				stDrag.mcMoveAbsolute.lrPosition		:= lrStartPositionTwoPhase;	
			END_IF	
	    	
			stDrag.mcMoveAbsolute.bExecute				:= TRUE;
        	
			IF stDrag.mcMoveAbsolute.bDone  THEN
				stDrag.mcMoveAbsolute.bExecute			:=	FALSE;
				eRunningState							:=	E_DragStationState.eLifting;
			END_IF                                      	                                              
		ELSIF bMoveToEndPosition AND NOT vis.bDosingTwoPhasesShow THEN
			stDrag.mcMoveAbsolute.lrPosition			:= lrEndPosition;
			stDrag.mcMoveAbsolute.bExecute				:= TRUE;
			eRunningState							:=	E_DragStationState.eLifting;
		ELSIF bMoveToEndPosition AND vis.bDosingTwoPhasesShow THEN
			stDrag.mcMoveAbsolute.lrPosition			:= lrEndPositionTwoPhase;
			stDrag.mcMoveAbsolute.bExecute				:= TRUE;
			eRunningState							:=	E_DragStationState.eLifting;	
		END_IF	
// Podnoszenie widel do przeciągania i sprawdzenie czy trafiły w otwór		
	E_DragStationState.eLifting:
	
		bDragActuator								:=	TRUE;		
		IF bDragUpSensor AND bRun THEN
			eRunningState							:=	E_DragStationState.eDraging;	
		END_IF
//  
	E_DragStationState.ePrepareToDrag:
		;
	
// Przeciąganie formatek
	E_DragStationState.eDraging:
	
		bLeadBefore1Actuator						:=	FALSE;	
		bLeadBefore2Actuator						:=	FALSE;
		
		IF NOT bTwoPhaseMode AND lrActualDragPosition > lrLeadActuatorMoveUpPosition THEN
			bLeadBefore1Actuator						:=	TRUE;	
		ELSIF bTwoPhaseMode AND lrActualDragPosition < (lrStartPositionTwoPhase - lrLeadActuatorMoveUpPosition) THEN
			bLeadBefore2Actuator						:=	TRUE;
		END_IF
			IF tonRunningDraging.Q THEN //100MS
				//Dynamika Ruchu
				stDrag.mcMoveAbsolute.lrAcceleration		:= lrDragAcceleration;
				stDrag.mcMoveAbsolute.lrDeceleration		:= lrDragDeceleration;
				stDrag.mcMoveAbsolute.lrJerk				:= lrDragJerk;
				stDrag.mcMoveAbsolute.lrVelocity			:= lrDragSpeed;
				
				IF NOT bMoveToEndPosition THEN
					stDrag.mcMoveAbsolute.lrPosition			:= lrMiddlePosition;
					IF bTwoPhaseMode THEN //dwu-faza
						stDrag.mcMoveAbsolute.lrPosition		:= lrMiddlePositionTwoPhase;	
					END_IF	
					stDrag.mcMoveAbsolute.bExecute				:= TRUE;
					IF stDrag.mcMoveAbsolute.bDone THEN
						stDrag.mcMoveAbsolute.bExecute			:= FALSE;
						eRunningState							:= E_DragStationState.eDragingDone;
					END_IF
				END_IF
	    IF bMoveToEndPosition AND NOT vis.bDosingTwoPhasesShow	THEN
			stDrag.mcMoveAbsolute.lrPosition			:= lrEndPosition;
			stDrag.mcMoveAbsolute.bExecute				:= TRUE;	
			IF stDrag.mcMoveAbsolute.bDone THEN
				stDrag.mcMoveAbsolute.bExecute			:= FALSE;
				bCycleDone								:= TRUE;
				eRunningState							:= E_DragStationState.eReady;
			END_IF
		ELSIF bMoveToEndPosition AND vis.bDosingTwoPhasesShow	THEN
			stDrag.mcMoveAbsolute.lrPosition			:= lrEndPositionTwoPhase;			
            stDrag.mcMoveAbsolute.bExecute				:= TRUE;	
            IF stDrag.mcMoveAbsolute.bDone THEN
            	stDrag.mcMoveAbsolute.bExecute			:= FALSE;
            	bCycleDone								:= TRUE;
            	eRunningState							:= E_DragStationState.eReady;
	        END_IF
		END_IF
		END_IF
		//Szybsze otwieranie prowadzeń ZA o 2mm szybciej ZA szlaban chaczy
		IF NOT bTwoPhaseMode AND lrActualDragPosition > (lrMiddlePosition - 2) THEN
			bLeadBefore2Actuator						:=	NOT bBefore2ActuatorOff;	
		ELSIF bTwoPhaseMode AND lrActualDragPosition < (lrMiddlePositionTwoPhase + 2) THEN
			bLeadBefore1Actuator						:=	TRUE;
		END_IF				
		
	E_DragStationState.eDragingDone:

		bLeadBefore1Actuator						:=	TRUE;
		bLeadBefore2Actuator						:=	NOT bBefore2ActuatorOff;		
		eRunningState								:= E_DragStationState.eEndingOfDrag;
	
	E_DragStationState.eEndingOfDrag:
	
		//Dynamika Ruchu
		stDrag.mcMoveAbsolute.lrAcceleration		:= lrDragAcceleration;
		stDrag.mcMoveAbsolute.lrDeceleration		:= lrDragDeceleration;
		stDrag.mcMoveAbsolute.lrJerk				:= lrDragJerk;		
		stDrag.mcMoveAbsolute.lrVelocity			:= lrDragSpeed;
		
		stDrag.mcMoveAbsolute.lrPosition			:= lrEndPosition;
		IF bTwoPhaseMode THEN //dwu-faza			//	3 +	(143 - 137) = 3 + 6 = 9
			stDrag.mcMoveAbsolute.lrPosition		:= lrEndPositionTwoPhase;	
		END_IF	
		stDrag.mcMoveAbsolute.bExecute				:= TRUE;
		
		IF stDrag.mcMoveAbsolute.bDone THEN
			
		 IF tonRunningeEndingOfDrag.Q OR NOT bDelayAfterDrag THEN //Opóżnienie na końcu ruchu z wysunietymi widłami
			stDrag.mcMoveAbsolute.bExecute			:= FALSE;
			eRunningState							:= E_DragStationState.eEndingOfDragDone;
		END_IF	
			
		END_IF
		
	E_DragStationState.eEndingOfDragDone:
		
		eRunningState								:= E_DragStationState.eLowering;
	
	E_DragStationState.eLowering:
	
		bDragActuator								:=	FALSE;		
		IF bDragDownSensor (*tonNotDragActuatorDelay.Q*) THEN
			eRunningState							:= E_DragStationState.eDraged;
		END_IF		

		
	E_DragStationState.eDraged:
	
		stDrag.mcMoveAbsolute.lrAcceleration		:= lrDragAcceleration;
		stDrag.mcMoveAbsolute.lrDeceleration		:= lrDragDeceleration;
		stDrag.mcMoveAbsolute.lrJerk				:= lrDragJerk;		
		stDrag.mcMoveAbsolute.lrVelocity			:= lrDragSpeed;
		
		stDrag.mcMoveAbsolute.lrPosition			:= lrStartPosition;
		IF bTwoPhaseMode THEN //dwu-faza			
			stDrag.mcMoveAbsolute.lrPosition		:= lrStartPositionTwoPhase;
		END_IF			
		
		stDrag.mcMoveAbsolute.bExecute				:= TRUE;
	
		IF stDrag.mcMoveAbsolute.bDone THEN
			stDrag.mcMoveAbsolute.bExecute			:= FALSE;
			eRunningState							:= E_DragStationState.eDragedDone;
		END_IF
		
	E_DragStationState.eDragedDone:
	
		bCycleDone									:= TRUE;	
		eRunningState								:= E_DragStationState.eReady;	
		
END_CASE
END_ACTION

ACTION Signals:

tonPreparingToReady		(IN:=	eState = E_Station.ePreparingToReady			,PT:= T#3S);
tonResetting			(IN:=	eState = E_Station.eResetting					,PT:= T#200MS);
tonHoming				(IN:=	eState = E_Station.eHoming						,PT:= T#1S);
rtResetCommands			(CLK:=	eState = E_Station.eReady 						,Q=>); 

tonRunningDraging		(IN:=	eRunningState = E_DragStationState.eDraging		,PT:= T#100MS);	//bylo 100
tonRunningeEndingOfDrag	(IN:=	eRunningState = E_DragStationState.eEndingOfDrag AND
								stDrag.mcMoveAbsolute.bDone
								,PT:= T#5MS);								//100ms t#200ms

//Opóżnienie wysuwania przeciągania
tonNotDragActuatorDelay	(IN:=	NOT bDragActuator					,PT:=T#150MS);

	
//Aktualna pozycja przeciągania
lrActualDragPosition:= stDrag.stStatus.lrActPos;


//
END_ACTION

ACTION Statistics:
rtrigCycleTimerRead(CLK:=bCycleDone);
IF rtrigCycleTimerRead.Q THEN
	tCycleTime:=tonCycleTimer.ET;
END_IF
tonCycleTimer(IN:= eRunningState>E_DragStationState.eReady, PT:=T#1D);
END_ACTION

END_FUNCTION_BLOCK

// ---- POUs/FB/POUsAxisOnline/NC/FB_McAxisOnlineNC.TcPOU
//==================================================================================================
//							Beckhoff Automation Poland
//									10.01.2019
//	Wszystkomajacy blok funkcyjny do sterowania osia, 
//	wymagane biblioteki: Tc2_MC2, Tc2_Utilities
// 	v1.0 	|| TC v 3.1.4022.27	 	|| - first edition
//==================================================================================================
{attribute 'reflection'}
FUNCTION_BLOCK FB_McAxisOnlineNC
VAR_IN_OUT
	stMcAxisOnline						: ST_McAxisOnline;
	Axis								: AXIS_REF;
END_VAR
VAR
	mcPower								: MC_Power;
	mcStop								: MC_Stop;
	mcHalt								: MC_Halt;
	mcStopSS1							: MC_Stop;
	mcStopSS2							: MC_Stop;
	mcReset								: MC_Reset;
	mcHome								: MC_Home;
	mcSetPosition						: MC_SetPosition;
	mcJog								: MC_Jog;

	mcMoveAbsolute						: MC_MoveAbsolute;
	mcMoveRelative						: MC_MoveRelative;
	mcMoveVelocity						: MC_MoveVelocity;
	mcMoveModulo						: MC_MoveModulo;
	mcMoveAbsolute2						: MC_MoveAbsolute;
	mcMoveRelative2						: MC_MoveRelative;
	mcMoveVelocity2						: MC_MoveVelocity;
	mcMoveModulo2						: MC_MoveModulo;

	fbNcLimitSwitch						: FB_NcSWLimitSwitchCtrl;
	mcReadParameterSet					: MC_ReadParameterSet;
	// Internal
	bInitialized						: BOOL;
			
	// Initialization
	iInitStep							: INT;
	bInitializationError				: BOOL;
	wInitializationErrorCounter			: WORD;
	bReadParameterSetReady				: BOOL;
	tonDelay							: TON;
	// Re init
	udiOnlineChangeCntOld				: UDINT;
	bOnlineChangeDetected				: BOOL;
	bReInit								: BOOL;
	bReInitialized						: BOOL;
	bReInitializationError				: BOOL;
	{attribute 'instance-path'}
	{attribute 'noinit'}
	sInstancePath						: STRING;
END_VAR

// Device dependent initialization 
ACT_Initialization();
// Device independent commands, mostly NC 
ACT_States();
ACT_SWLimitSwitch();
ACT_Stop();
ACT_Power();
ACT_Homing();
ACT_Jog();
ACT_Move();
ACT_ResetAndDiag();
ACT_SetPosition();
// Device independent error collection
ACT_ErrorCollection();

ACTION ACT_ErrorCollection:
// Error flags
stMcAxisOnline.stError.bDriveError					:= Axis.Status.DriveDeviceError;

stMcAxisOnline.stError.bNcError						:= Axis.Status.Error;

stMcAxisOnline.stError.bFBError						:= stMcAxisOnline.mcPower.bError OR stMcAxisOnline.mcReset.bError OR stMcAxisOnline.mcHome.bError OR stMcAxisOnline.mcJog.bError
													OR stMcAxisOnline.mcHalt.bError OR stMcAxisOnline.mcStop.bError OR stMcAxisOnline.mcSS1.bError OR stMcAxisOnline.mcSS2.bError
													OR stMcAxisOnline.mcMoveAbsolute.bError OR stMcAxisOnline.mcMoveRelative.bError OR stMcAxisOnline.mcMoveVelocity.bError OR stMcAxisOnline.mcMoveModulo.bError
													OR stMcAxisOnline.mcMoveAbsolute2.bError OR stMcAxisOnline.mcMoveRelative2.bError OR stMcAxisOnline.mcMoveVelocity2.bError OR stMcAxisOnline.mcMoveModulo2.bError
													OR stMcAxisOnline.stNcLimitSwitch.bError OR stMcAxisOnline.mcSetPosition.bError;
									
stMcAxisOnline.stError.bCommunicationError			:= stMcAxisOnline.stChannelErrorCode.bError OR stMcAxisOnline.stSetPositionOffset.bError OR stMcAxisOnline.stMotorMonitoring.bError OR stMcAxisOnline.stHoldingBrake.bError;

stMcAxisOnline.stError.bError						:= stMcAxisOnline.stError.bDriveError OR stMcAxisOnline.stError.bNcError OR stMcAxisOnline.stError.bFBError OR stMcAxisOnline.stError.bCommunicationError;
stMcAxisOnline.bError								:= stMcAxisOnline.stError.bError; // Forward one stage up

// Error codes
stMcAxisOnline.stError.uiDriveErrorID 				:= stMcAxisOnline.stChannelErrorCode.uiChannelErrorCode;
stMcAxisOnline.stError.uiDriveErrorIDHex 			:= stMcAxisOnline.stChannelErrorCode.uiChannelErrorCodeHex;

stMcAxisOnline.stError.udiNcErrorID 				:= Axis.Status.ErrorID;
stMcAxisOnline.stError.udiNcErrorIDHex 				:= Axis.Status.ErrorID;
	

stMcAxisOnline.stError.udiFBErrorID 				:= 	stMcAxisOnline.mcPower.udiErrorID + 
														stMcAxisOnline.mcReset.udiErrorID + 
														stMcAxisOnline.mcHome.udiErrorID + 
														stMcAxisOnline.mcJog.udiErrorID +
														stMcAxisOnline.mcHalt.udiErrorID + 
														stMcAxisOnline.mcStop.udiErrorID + 
														stMcAxisOnline.mcSS1.udiErrorID + 
														stMcAxisOnline.mcSS2.udiErrorID +
														stMcAxisOnline.mcMoveAbsolute.udiErrorID + 
														stMcAxisOnline.mcMoveRelative.udiErrorID + 
														stMcAxisOnline.mcMoveVelocity.udiErrorID + 
														stMcAxisOnline.mcMoveModulo.udiErrorID +
														stMcAxisOnline.mcMoveAbsolute2.udiErrorID + 
														stMcAxisOnline.mcMoveRelative2.udiErrorID + 
														stMcAxisOnline.mcMoveVelocity2.udiErrorID + 
														stMcAxisOnline.mcMoveModulo2.udiErrorID +
														stMcAxisOnline.stNcLimitSwitch.udiErrorID + 
														stMcAxisOnline.mcSetPosition.udiErrorID;

stMcAxisOnline.stError.udiFBErrorIDHex 				:= stMcAxisOnline.stError.udiFBErrorID;

stMcAxisOnline.stError.udiErrorID					:= stMcAxisOnline.stSetPositionOffset.udiErrorID;
stMcAxisOnline.stError.uiAdsErrorID					:= stMcAxisOnline.stChannelErrorCode.uiAdsErrId + stMcAxisOnline.stMotorMonitoring.uiAdsErrId + stMcAxisOnline.stHoldingBrake.uiAdsErrId;
stMcAxisOnline.stError.uiSecErrorID					:= stMcAxisOnline.stChannelErrorCode.uiSecErrId + stMcAxisOnline.stMotorMonitoring.uiSecErrId + stMcAxisOnline.stHoldingBrake.uiSecErrId;

stMcAxisOnline.stError.sNcError						:= F_AxErrMsg(stMcAxisOnline.stError.udiNcErrorID);
stMcAxisOnline.stError.sDriveError					:= F_AX5xErrMsg(stMcAxisOnline.stError.uiDriveErrorID);
END_ACTION

ACTION ACT_Homing:
mcHome(		Axis						:= Axis,
			Execute						:= stMcAxisOnline.mcHome.bExecute,
			Position					:= stMcAxisOnline.mcHome.lrPosition,
			HomingMode					:= stMcAxisOnline.mcHome.eHomingMode,
			BufferMode					:= stMcAxisOnline.mcHome.eBufferMode,
			Options						:= stMcAxisOnline.mcHome.stOptions,
			bCalibrationCam				:= stMcAxisOnline.mcHome.bCalibrationCam,
			Done						=> stMcAxisOnline.mcHome.bDone,
			Busy						=> stMcAxisOnline.mcHome.bBusy,
			Active						=> stMcAxisOnline.mcHome.bActive,
			CommandAborted				=> stMcAxisOnline.mcHome.bCommandAborted,
			Error						=> stMcAxisOnline.mcHome.bError,
			ErrorID						=> stMcAxisOnline.mcHome.udiErrorID);
END_ACTION

ACTION ACT_Initialization:
// bInitialized flag is set just once. 
// bReInitialized ise set each time we do online change or request reinit operation
// bDriveAddressReady, bReadParameterSetReady, bDriveRefReady - set just once after successed read

// Online change detection
bOnlineChangeDetected					:= udiOnlineChangeCntOld <> _AppInfo.OnlineChangeCnt;
udiOnlineChangeCntOld 					:= _AppInfo.OnlineChangeCnt;
// Reset init
IF bReInit OR bOnlineChangeDetected THEN
	iInitStep							:= 0;
END_IF

//Initialization process
CASE iInitStep OF
	0:	// Read Parameter Set
		
		stMcAxisOnline.mcReadParameterSet.bExecute		:=	 TRUE;
		iInitStep						:= iInitStep + 10;
		
	10: // Wait for data
	
		IF NOT stMcAxisOnline.mcReadParameterSet.bBusy THEN
			stMcAxisOnline.mcReadParameterSet.bExecute	:=	 FALSE;
			IF stMcAxisOnline.mcReadParameterSet.bDone THEN
				iInitStep 				:= iInitStep + 10;
				bReadParameterSetReady 	:= TRUE;
			ELSE
				iInitStep 				:= 1000;		// Error step
			END_IF
		END_IF	
	
	20: // Success - initialized flag, clear error
		bReInitialized					:= bInitialized;	// TRUE only when it's not first initialization e.g. online change
		bInitialized 					:= TRUE;
		bReInitializationError			:= FALSE;			// TRUE only when it's not first initialization e.g. online change
		bInitializationError			:= FALSE;
		iInitStep 						:= iInitStep + 10;
		
	30: // Idle
	
		;
		
	1000: // Error step
		wInitializationErrorCounter 	:= wInitializationErrorCounter + 1;
		IF wInitializationErrorCounter < 100 THEN
			iInitStep					:= iInitStep + 5;			// Go to delay
		ELSE
			bReInitializationError		:= bInitializationError;	// TRUE only when it's not first initialization e.g. online change
			bInitializationError		:= TRUE;
			bReInitialized				:= FALSE;
			iInitStep 					:= iInitStep + 10;
		END_IF

	1005: // Delay step
		tonDelay(IN:= TRUE, PT:= T#1S);
		IF tonDelay.Q THEN
			tonDelay(IN:= FALSE, PT:= T#1S);
			iInitStep					:= 0;
		END_IF
		
	1010: // Idle after error
		;
	
END_CASE
				
mcReadParameterSet(	Parameter			:= stMcAxisOnline.stAxisParameter,
					Axis				:= Axis,
					Execute				:= stMcAxisOnline.mcReadParameterSet.bExecute,
					Done				=> stMcAxisOnline.mcReadParameterSet.bDone,
					Busy				=> stMcAxisOnline.mcReadParameterSet.bBusy,
					Error				=> stMcAxisOnline.mcReadParameterSet.bError,
					ErrorID				=> stMcAxisOnline.mcReadParameterSet.udiErrorID);
END_ACTION

ACTION ACT_Jog:
// Direct access from bSlow or bFast, if none then free choice
IF stMcAxisOnline.mcJog.bSlowForward OR stMcAxisOnline.mcJog.bSlowBackward THEN
	stMcAxisOnline.mcJog.eMode			:= MC_JOGMODE_STANDARD_SLOW;
ELSIF stMcAxisOnline.mcJog.bFastForward OR stMcAxisOnline.mcJog.bFastBackward THEN
	stMcAxisOnline.mcJog.eMode			:= MC_JOGMODE_STANDARD_FAST;
END_IF

mcJog(		Axis						:= Axis,
			JogForward					:= stMcAxisOnline.mcJog.bJogForward OR stMcAxisOnline.mcJog.bSlowForward OR stMcAxisOnline.mcJog.bFastForward,
			JogBackwards				:= stMcAxisOnline.mcJog.bJogBackwards OR stMcAxisOnline.mcJog.bSlowBackward OR stMcAxisOnline.mcJog.bFastBackward,
			Mode						:= stMcAxisOnline.mcJog.eMode,
			Position					:= stMcAxisOnline.mcJog.lrPosition,
			Velocity					:= stMcAxisOnline.mcJog.lrVelocity,
			Acceleration				:= stMcAxisOnline.mcJog.lrAcceleration,
			Deceleration				:= stMcAxisOnline.mcJog.lrDeceleration,
			Jerk						:= stMcAxisOnline.mcJog.lrJerk,
			Done						=> stMcAxisOnline.mcJog.bDone,
			Busy						=> stMcAxisOnline.mcJog.bBusy,
			Active						=> stMcAxisOnline.mcJog.bActive,
			CommandAborted				=> stMcAxisOnline.mcJog.bCommandAborted,
			Error						=> stMcAxisOnline.mcJog.bError,
			ErrorID						=> stMcAxisOnline.mcJog.udiErrorID);
END_ACTION

ACTION ACT_Move:
{region "Primary"}
mcMoveAbsolute(	Axis					:= Axis,
				Execute					:= stMcAxisOnline.mcMoveAbsolute.bExecute,
				Position				:= stMcAxisOnline.mcMoveAbsolute.lrPosition,
				Velocity				:= stMcAxisOnline.mcMoveAbsolute.lrVelocity,
				Acceleration			:= stMcAxisOnline.mcMoveAbsolute.lrAcceleration,
				Deceleration			:= stMcAxisOnline.mcMoveAbsolute.lrDeceleration,
				Jerk					:= stMcAxisOnline.mcMoveAbsolute.lrJerk,
				BufferMode				:= stMcAxisOnline.mcMoveAbsolute.eBufferMode,
				Options					:= stMcAxisOnline.mcMoveAbsolute.stOptions,
				Done					=> stMcAxisOnline.mcMoveAbsolute.bDone,
				Busy					=> stMcAxisOnline.mcMoveAbsolute.bBusy,
				Active					=> stMcAxisOnline.mcMoveAbsolute.bActive,
				CommandAborted			=> stMcAxisOnline.mcMoveAbsolute.bCommandAborted,
				Error					=> stMcAxisOnline.mcMoveAbsolute.bError,
				ErrorID					=> stMcAxisOnline.mcMoveAbsolute.udiErrorID);

mcMoveRelative(	Axis					:= Axis,
				Execute					:= stMcAxisOnline.mcMoveRelative.bExecute,
				Distance				:= stMcAxisOnline.mcMoveRelative.lrDistance,
				Velocity				:= stMcAxisOnline.mcMoveRelative.lrVelocity,
				Acceleration			:= stMcAxisOnline.mcMoveRelative.lrAcceleration,
				Deceleration			:= stMcAxisOnline.mcMoveRelative.lrDeceleration,
				Jerk					:= stMcAxisOnline.mcMoveRelative.lrJerk,
				BufferMode				:= stMcAxisOnline.mcMoveRelative.eBufferMode,
				Options					:= stMcAxisOnline.mcMoveRelative.stOptions,
				Done					=> stMcAxisOnline.mcMoveRelative.bDone,
				Busy					=> stMcAxisOnline.mcMoveRelative.bBusy,
				Active					=> stMcAxisOnline.mcMoveRelative.bActive,
				CommandAborted			=> stMcAxisOnline.mcMoveRelative.bCommandAborted,
				Error					=> stMcAxisOnline.mcMoveRelative.bError,
				ErrorID					=> stMcAxisOnline.mcMoveRelative.udiErrorID);
				
mcMoveVelocity(	Axis					:= Axis,
				Execute					:= stMcAxisOnline.mcMoveVelocity.bExecute,
				Velocity				:= stMcAxisOnline.mcMoveVelocity.lrVelocity,
				Acceleration			:= stMcAxisOnline.mcMoveVelocity.lrAcceleration,
				Deceleration			:= stMcAxisOnline.mcMoveVelocity.lrDeceleration,
				Jerk					:= stMcAxisOnline.mcMoveVelocity.lrJerk,
				Direction				:= stMcAxisOnline.mcMoveVelocity.eDirection,
				BufferMode				:= stMcAxisOnline.mcMoveVelocity.eBufferMode,
				Options					:= stMcAxisOnline.mcMoveVelocity.stOptions,
				InVelocity				=> stMcAxisOnline.mcMoveVelocity.bInVelocity,
				Busy					=> stMcAxisOnline.mcMoveVelocity.bBusy,
				Active					=> stMcAxisOnline.mcMoveVelocity.bActive,
				CommandAborted			=> stMcAxisOnline.mcMoveVelocity.bCommandAborted,
				Error					=> stMcAxisOnline.mcMoveVelocity.bError,
				ErrorID					=> stMcAxisOnline.mcMoveVelocity.udiErrorID);
stMcAxisOnline.mcMoveVelocity.bDone		:= stMcAxisOnline.mcMoveVelocity.bInVelocity;

mcMoveModulo(	Axis					:= Axis,
				Execute					:= stMcAxisOnline.mcMoveModulo.bExecute,
				Position				:= stMcAxisOnline.mcMoveModulo.lrPosition,
				Velocity				:= stMcAxisOnline.mcMoveModulo.lrVelocity,
				Acceleration			:= stMcAxisOnline.mcMoveModulo.lrAcceleration,
				Deceleration			:= stMcAxisOnline.mcMoveModulo.lrDeceleration,
				Jerk					:= stMcAxisOnline.mcMoveModulo.lrJerk,
				Direction				:= stMcAxisOnline.mcMoveModulo.eDirection,
				BufferMode				:= stMcAxisOnline.mcMoveModulo.eBufferMode,
				Options					:= stMcAxisOnline.mcMoveModulo.stOptions,
				Done					=> stMcAxisOnline.mcMoveModulo.bDone,
				Busy					=> stMcAxisOnline.mcMoveModulo.bBusy,
				Active					=> stMcAxisOnline.mcMoveModulo.bActive,
				CommandAborted			=> stMcAxisOnline.mcMoveModulo.bCommandAborted,
				Error					=> stMcAxisOnline.mcMoveModulo.bError,
				ErrorID					=> stMcAxisOnline.mcMoveModulo.udiErrorID);
{endregion}
{region "Secondary"}
mcMoveAbsolute2(Axis					:= Axis,
				Execute					:= stMcAxisOnline.mcMoveAbsolute2.bExecute,
				Position				:= stMcAxisOnline.mcMoveAbsolute2.lrPosition,
				Velocity				:= stMcAxisOnline.mcMoveAbsolute2.lrVelocity,
				Acceleration			:= stMcAxisOnline.mcMoveAbsolute2.lrAcceleration,
				Deceleration			:= stMcAxisOnline.mcMoveAbsolute2.lrDeceleration,
				Jerk					:= stMcAxisOnline.mcMoveAbsolute2.lrJerk,
				BufferMode				:= stMcAxisOnline.mcMoveAbsolute2.eBufferMode,
				Options					:= stMcAxisOnline.mcMoveAbsolute2.stOptions,
				Done					=> stMcAxisOnline.mcMoveAbsolute2.bDone,
				Busy					=> stMcAxisOnline.mcMoveAbsolute2.bBusy,
				Active					=> stMcAxisOnline.mcMoveAbsolute2.bActive,
				CommandAborted			=> stMcAxisOnline.mcMoveAbsolute2.bCommandAborted,
				Error					=> stMcAxisOnline.mcMoveAbsolute2.bError,
				ErrorID					=> stMcAxisOnline.mcMoveAbsolute2.udiErrorID);

